// TIA Portal project "TFG_MaiteLopez" (V16)

(* hardware
DEVICE "S71500/ET200MP station_1"  S7-1500 station
   slot 0: "Perfil soporte_0"  Rack  6ES7 590-1***0-0AA0
   slot 1: "PLC_1"  CPU 1513-1 PN  6ES7 513-1AL01-0AB0  V2.8
      slot 3: "Display de la CPU_1"  6ES7591-1AA00-0AA0
      slot 32768: "Interfaz PROFINET_1"  X1
         slot 32769: "Puerto_1"  X1 P1
         slot 32770: "Puerto_2"  X1 P2
      slot 34817: "Virtual CP interface port_1"  Virtual CP interface port  Virtual CP interface port
DEVICE "HMI_1"  KTP400 Basic PN
   slot 0: "HMI_1"  KTP400 Basic PN  6AV2 123-2DB03-0AX0  16.0.0.0
   slot 1: "HMI_RT_1"  KTP400 Basic PN  6AV2 123-2DB03-0AX0  16.0.0.0
   slot 5: "HMI_1.IE_CP_1"  PROFINET Interface  16.0.0.0
      slot 1: "Interfaz PROFINET_1"  PROFINET Interface
         slot 1: "Port_1"  Port
*)

// ===== PLC "PLC_1"  CPU 1513-1 PN =====

VAR_GLOBAL   // PLC tag table "Entradas"
   "FactoryIO_Reseting" AT %I1.6 : Bool;
   "FactoryIO_Running" AT %I1.7 : Bool;
   "AtEntry" AT %I0.0 : Bool;
   "AtLoad" AT %I0.1 : Bool;
   "AtLeft" AT %I0.2 : Bool;
   "AtMiddle" AT %I0.3 : Bool;
   "AtRight" AT %I0.4 : Bool;
   "AtUnload" AT %I0.5 : Bool;
   "AtExit" AT %I0.6 : Bool;
   "MovingX" AT %I0.7 : Bool;
   "MovingZ" AT %I1.0 : Bool;
END_VAR

VAR_GLOBAL   // PLC tag table "HMI"
   "Marcha" AT %M5.0 : Bool;
   "Paro" AT %M5.1 : Bool;
   "Reset" AT %M5.2 : Bool;
   "AutoMan" AT %M5.3 : Bool;
   "Posicion" AT %MW8 : Int;
   "Men1" AT %M10.0 : Bool;
   "Men2" AT %M10.1 : Bool;
   "Men3" AT %M10.2 : Bool;
   "Emergencia" AT %M10.3 : Bool;
   "AuxMarcha" AT %M10.4 : Bool;
   "AuxParo" AT %M10.5 : Bool;
END_VAR

VAR_GLOBAL   // PLC tag table "Salidas"
   "TargetPosition" AT %QW2 : Word;
   "EntryConveyor" AT %Q0.0 : Bool;
   "LoadConveyor" AT %Q0.1 : Bool;
   "ForksLeft" AT %Q0.2 : Bool;
   "ForksRight" AT %Q0.3 : Bool;
   "Lift" AT %Q0.4 : Bool;
   "UnloadConveyor" AT %Q0.5 : Bool;
   "ExitConveyor" AT %Q0.6 : Bool;
   "Emitter" AT %Q1.2 : Bool;
   "Remover" AT %Q1.3 : Bool;
   "FactoryIO_Reset" AT %Q1.4 : Bool;
   "FactoryIO_Run" AT %Q1.5 : Bool;
END_VAR

VAR_GLOBAL   // PLC tag table "Señales de Control"
   "Inicio" AT %M0.0 : Bool;
   "SolCondIni" AT %M0.1 : Bool;
   "FinCondIni" AT %M0.2 : Bool;
   "ProdNorm" AT %M0.3 : Bool;
   "ParoFC" AT %M0.4 : Bool;
   "DejarCoger" AT %M0.5 : Bool;
   "FinDejar" AT %M0.7 : Bool;
   "InitGraf" AT %M1.6 : Bool;
   "ResetGraf" AT %M1.7 : Bool;
   "AuxInit" AT %M2.0 : Bool;
   "SolDejar" AT %M0.6 : Bool;
   "SolEntradaMaterial" AT %M1.2 : Bool;
   "FinEntradaMaterial" AT %M1.3 : Bool;
   "SolSalidaMaterial" AT %M1.4 : Bool;
   "FinSalidaMaterial" AT %M1.5 : Bool;
   "SolCoger" AT %M1.0 : Bool;
   "FinCoger" AT %M1.1 : Bool;
   "InicializarAlmacenOcupacion" AT %M2.1 : Bool;
END_VAR

DATA_BLOCK "Sensores"   // DB1
{ S7_Optimized_Access := 'FALSE' }
VERSION : 0.1
   VAR
      AlmacenOcupacion : Array[1..54] of Bool;
   END_VAR
BEGIN
END_DATA_BLOCK

DATA_BLOCK "CogerDejar_DB"   // DB2
{ S7_Optimized_Access := 'TRUE' }
VERSION : 0.1
// stored: InstanceOfName GCogerDejar
"GCogerDejar"
BEGIN
END_DATA_BLOCK

DATA_BLOCK "CondIniciales_DB"   // DB4
{ S7_Optimized_Access := 'TRUE' }
VERSION : 0.1
// stored: InstanceOfName GCondIniciales
"GCondIniciales"
BEGIN
END_DATA_BLOCK

DATA_BLOCK "MaterialIO_DB"   // DB5
{ S7_Optimized_Access := 'TRUE' }
VERSION : 0.1
// stored: InstanceOfName GMaterialIO
"GMaterialIO"
BEGIN
END_DATA_BLOCK

DATA_BLOCK "Emergencia_DB"   // DB6
{ S7_Optimized_Access := 'TRUE' }
VERSION : 0.1
// stored: InstanceOfName GEmergencia
"GEmergencia"
BEGIN
END_DATA_BLOCK

DATA_BLOCK "DB_OPCUA"   // DB7
{ S7_Optimized_Access := 'TRUE' }
VERSION : 0.1
   VAR
      control_parameters : Struct
         Control_Flag_New_Service : Bool := false;
         Control_Flag_Item_Completed : Bool;
         Control_Flag_Service_Completed : Bool;
      END_STRUCT;
      data_from_GW : Struct
         Id_Machine_Reference : UDInt;
         Id_Order_Reference : UDInt;
         Id_Batch_Reference : UDInt;
         Operation_Ref_Service_Type : UDInt := 1;
         Operation_No_of_Items : UDInt := 4;
      END_STRUCT;
      data_to_GW : Struct
         Id_Machine_Reference : UDInt;
         Id_Order_Reference : UDInt;
         Id_Batch_Reference : UDInt;
         Id_Ref_Service_Type : UDInt;
         Id_Item_Number : USInt;
         Data_Initial_Time_Stamp : String;
         Data_Final_Time_Stamp_1 : String;
         Data_Service_Time_Stamp : String;
      END_STRUCT;
   END_VAR
BEGIN
END_DATA_BLOCK

DATA_BLOCK "GestionarAlmacen_DB"   // DB8
{ S7_Optimized_Access := 'TRUE' }
VERSION : 0.1
// stored: InstanceOfName GGestionarAlmacen
"GGestionarAlmacen"
BEGIN
END_DATA_BLOCK

DATA_BLOCK "SecPrincipal_ST_DB"   // DB9
{ S7_Optimized_Access := 'TRUE' }
VERSION : 0.1
// stored: InstanceOfName GSecPrincipal_ST
"GSecPrincipal_ST"
BEGIN
END_DATA_BLOCK

// folder: System blocks/Program resources

DATA_BLOCK "IEC_Timer_0_DB"   // DB3
{ S7_Optimized_Access := 'TRUE' }
AUTHOR : Simatic
FAMILY : IEC
NAME : IEC_TMR
VERSION : 1.0
// stored: InstanceOfName IEC_TIMER
"IEC_TIMER"
BEGIN
END_DATA_BLOCK

DATA_BLOCK "Interfaz del cliente_1_Configuration"   // DB10
{ S7_Optimized_Access := 'TRUE' }
   VAR
      Connection : Struct
         ConnectInfo : OPC_UA_SessionConnectInfo;
         ConnectionHdl : DWord;
         ServerEndpointUrl : String[254] := 'opc.tcp://:4840';
      END_STRUCT;
      Namespaces : Struct
         NamespaceURIs : Array[0..0] of WString;
         ServerNamespaceIndexes : Array[0..0] of UInt;
         NamespaceStatusList : Array[0..0] of DWord;
         NamespaceCount : UInt := 0;
      END_STRUCT;
   END_VAR
BEGIN
   Connection.ConnectInfo.SessionName := WSTRING#'Conexión OPC UA_1';
   Connection.ConnectInfo.ApplicationName := WSTRING#'';
   Connection.ConnectInfo.SecurityMsgMode := 1;
   Connection.ConnectInfo.SecurityPolicy := 1;
   Connection.ConnectInfo.CheckServerCertificate := False;
   Connection.ConnectInfo.TransportProfile := 1;
   Connection.ConnectInfo.UserIdentityTokenType := 0;
   Connection.ConnectInfo.CertificateID := 0;
   Connection.ConnectInfo.SessionTimeout := T#30S;
   Connection.ConnectInfo.MonitorConnection := T#5S;
   Connection.ConnectInfo.LocaleIDs[0] := 'es-ES';
   Connection.ConnectInfo.LocaleIDs[1] := '';
   Connection.ConnectInfo.LocaleIDs[2] := '';
   Connection.ConnectInfo.LocaleIDs[3] := '';
   Connection.ConnectInfo.LocaleIDs[4] := '';
END_DATA_BLOCK

// folder: (top level)

FUNCTION_BLOCK "GGestionarAlmacen"   // FB1, GRAPH_PLUS
{ S7_Optimized_Access := 'TRUE' }
VERSION : 0.1
   VAR_INPUT
      OFF_SQ : Bool := false;   // Desactivar cadena
      INIT_SQ : Bool := false;   // Poner cadena en estado inicial
      ACK_EF : Bool := false;   // Acusar todos los errores y fallos
      S_PREV : Bool := false;   // Mostrar la etapa anterior en el parámetro S_NO
      S_NEXT : Bool := false;   // Mostrar la etapa siguiente en el parámetro S_NO
      SW_AUTO : Bool := false;   // Modo automático
      SW_TAP : Bool := false;   // Semiautomático/continuar con transición
      SW_TOP : Bool := false;   // Semiautomático/transición ignorada
      SW_MAN : Bool := false;   // Modo manual
      S_SEL : Int := 0;   // Seleccionar la etapa que debe mostrarse en S_NO
      S_ON : Bool := false;   // Activar la etapa del parámetro S_NO
      S_OFF : Bool := false;   // Desactivar el incremento presente en el parámetro S_NO
      T_PUSH : Bool := false;   // Habilitar conmutación de transición en modo semiautomático
   END_VAR
   VAR_OUTPUT
      S_NO : Int := 0;   // Número de etapa
      S_MORE : Bool := false;   // Existen más etapas que pueden mostrarse en S_NO.
      S_ACTIVE : Bool := false;   // El incremento presente en el parámetro S_NO está activo
      ERR_FLT : Bool := false;   // Error de grupo interlock o supervisión
      AUTO_ON : Bool := false;   // Modo automático activado
      TAP_ON : Bool := false;   // Modo semiautomático/etapa con transición activada
      TOP_ON : Bool := false;   // Modo semiautomático/Ignorar transición activado
      MAN_ON : Bool := false;   // Modo manual activado
   END_VAR
   VAR
      HMI_INFO : Array[0..8] of UInt;
      IF_PAR : G7_IfParPlus_V4;
      RT_DATA : G7_RTDataPlus_V4;   // Área de datos interna
      Trans1 : G7_TransitionPlus_V4;   // Estructura de la transición
      Trans2 : G7_TransitionPlus_V4;   // Estructura de la transición
      Trans3 : G7_TransitionPlus_V4;   // Estructura de la transición
      Trans4 : G7_TransitionPlus_V4;   // Estructura de la transición
      Trans5 : G7_TransitionPlus_V4;   // Estructura de la transición
      Trans6 : G7_TransitionPlus_V4;   // Estructura de la transición
      Trans7 : G7_TransitionPlus_V4;   // Estructura de la transición
      Trans8 : G7_TransitionPlus_V4;   // Estructura de la transición
      Trans9 : G7_TransitionPlus_V4;   // Estructura de la transición
      Trans10 : G7_TransitionPlus_V4;   // Estructura de la transición
      Trans11 : G7_TransitionPlus_V4;   // Estructura de la transición
      Trans12 : G7_TransitionPlus_V4;   // Estructura de la transición
      Trans14 : G7_TransitionPlus_V4;   // Estructura de la transición
      Trans18 : G7_TransitionPlus_V4;   // Estructura de la transición
      Trans19 : G7_TransitionPlus_V4;   // Estructura de la transición
      Trans26 : G7_TransitionPlus_V4;   // Estructura de la transición
      Trans27 : G7_TransitionPlus_V4;   // Estructura de la transición
      Trans28 : G7_TransitionPlus_V4;   // Estructura de la transición
      Trans29 : G7_TransitionPlus_V4;   // Estructura de la transición
      Trans30 : G7_TransitionPlus_V4;   // Estructura de la transición
      Trans31 : G7_TransitionPlus_V4;   // Estructura de la transición
      Trans32 : G7_TransitionPlus_V4;   // Estructura de la transición
      Trans35 : G7_TransitionPlus_V4;   // Estructura de la transición
      X40 : G7_StepPlus_V4;   // Estructura de la etapa
      X41 : G7_StepPlus_V4;   // Estructura de la etapa
      X42 : G7_StepPlus_V4;   // Estructura de la etapa
      X43 : G7_StepPlus_V4;   // Estructura de la etapa
      X44 : G7_StepPlus_V4;   // Estructura de la etapa
      X46 : G7_StepPlus_V4;   // Estructura de la etapa
      X47 : G7_StepPlus_V4;   // Estructura de la etapa
      X56 : G7_StepPlus_V4;   // Estructura de la etapa
      X57 : G7_StepPlus_V4;   // Estructura de la etapa
      X48 : G7_StepPlus_V4;   // Estructura de la etapa
      X49 : G7_StepPlus_V4;   // Estructura de la etapa
      X50 : G7_StepPlus_V4;   // Estructura de la etapa
      X52 : G7_StepPlus_V4;   // Estructura de la etapa
      X53 : G7_StepPlus_V4;   // Estructura de la etapa
      X54 : G7_StepPlus_V4;   // Estructura de la etapa
      X55 : G7_StepPlus_V4;   // Estructura de la etapa
      X51 : G7_StepPlus_V4;   // Estructura de la etapa
      X45 : G7_StepPlus_V4;   // Estructura de la etapa
      X58 : G7_StepPlus_V4;   // Estructura de la etapa
      SINI : Array[0..1] of USInt;
      LSTT : Array[0..22] of USInt;
      ATAJ : Array[0..22] of USInt;
      ATAB : Array[0..22] of USInt;
      PSTT : Array[0..22] of USInt;
      NSTT : Array[0..22] of USInt;
      ASSJ : Array[0..18] of USInt;
      ASSB : Array[0..18] of USInt;
      PTTS : Array[0..18] of USInt;
      NTTS : Array[0..18] of USInt;
      SW_SQTS : Array[0..18] of USInt;
      SWITCH : Array[0..6] of USInt;
      TVX : Array[0..8] of USInt;
      TTX : Array[0..8] of USInt;
      TSX : Array[0..1] of USInt;
      S00X : Array[0..1] of USInt;
      SOFFX : Array[0..1] of USInt;
      SONX : Array[0..1] of USInt;
      SAX : Array[0..1] of USInt;
      SERRX : Array[0..19] of USInt;
      SMX : Array[0..19] of USInt;
      S0X : Array[0..19] of USInt;
      S1X : Array[0..19] of USInt;
      IL_ALARM_INST : Diag_Alarm;
      SUP_ALARM_INST : Diag_Alarm;
      STEP_TIME_ALARM_INST : Diag_Alarm;
      IEC_TIMER_INST : IEC_TIMER;
      TRANSACTION_FLAG : Bool := false;
   END_VAR
   // SINI[0] := 2;
   // LSTT[0] := 255;
   // LSTT[1] := 255;
   // LSTT[2] := 255;
   // LSTT[3] := 255;
   // LSTT[4] := 255;
   // LSTT[5] := 255;
   // ATAJ[1] := 1;
   // ATAJ[2] := 2;
   // ATAJ[3] := 3;
   // ATAJ[4] := 4;
   // ATAJ[5] := 5;
   // ATAJ[6] := 6;
   // ATAB[1] := 7;
   // ATAB[2] := 8;
   // ATAB[3] := 12;
   // ATAB[4] := 4;
   // ATAB[5] := 5;
   // ATAB[6] := 6;
   // PSTT[1] := 1;
   // PSTT[2] := 2;
   // PSTT[3] := 3;
   // PSTT[4] := 4;
   // PSTT[5] := 5;
   // PSTT[6] := 6;
   // NSTT[0] := 1;
   // NSTT[1] := 2;
   // NSTT[2] := 3;
   // NSTT[3] := 4;
   // NSTT[4] := 17;
   // NSTT[5] := 6;
   // ASSJ[1] := 1;
   // ASSJ[2] := 2;
   // ASSJ[3] := 3;
   // ASSJ[4] := 4;
   // ASSJ[5] := 5;
   // ASSJ[6] := 6;
   // ASSB[1] := 1;
   // ASSB[2] := 2;
   // ASSB[3] := 3;
   // ASSB[4] := 4;
   // ASSB[5] := 5;
   // ASSB[6] := 6;
   // PTTS[0] := 255;
   // PTTS[2] := 1;
   // PTTS[3] := 2;
   // PTTS[4] := 3;
   // PTTS[5] := 21;
   // PTTS[6] := 5;
   // NTTS[1] := 1;
   // NTTS[2] := 2;
   // NTTS[3] := 3;
   // NTTS[4] := 4;
   // NTTS[5] := 5;
   // NTTS[6] := 6;
   // TVX[0] := 16#1;
   // TTX[0] := 16#1;
   // TSX[0] := 16#1;
   // S00X[0] := 16#1;
   // SOFFX[0] := 16#1;
   // SONX[0] := 16#1;
   // SAX[0] := 16#1;
   // SERRX[0] := 16#1;
   // SMX[0] := 16#1;
   // S0X[0] := 16#1;
   // S1X[0] := 16#1;
   // LSTT[6] := 255;
   // LSTT[8] := 255;
   // LSTT[9] := 255;
   // ATAJ[7] := 7;
   // ATAJ[8] := 8;
   // ATAJ[9] := 9;
   // ATAJ[10] := 10;
   // ATAJ[11] := 11;
   // ATAJ[12] := 12;
   // ATAB[7] := 1;
   // ATAB[8] := 9;
   // ATAB[9] := 2;
   // ATAB[10] := 10;
   // ATAB[11] := 11;
   // ATAB[12] := 3;
   // PSTT[7] := 1;
   // PSTT[8] := 2;
   // PSTT[9] := 2;
   // PSTT[10] := 7;
   // PSTT[11] := 8;
   // PSTT[12] := 3;
   // NSTT[6] := 9;
   // NSTT[8] := 7;
   // NSTT[9] := 8;
   // ASSJ[7] := 7;
   // ASSJ[8] := 8;
   // ASSJ[9] := 9;
   // ASSB[7] := 7;
   // ASSB[8] := 8;
   // ASSB[9] := 9;
   // PTTS[7] := 8;
   // PTTS[8] := 9;
   // PTTS[9] := 6;
   // NTTS[7] := 10;
   // NTTS[8] := 11;
   // NTTS[9] := 13;
   // SW_SQTS[2] := 1;
   // SW_SQTS[3] := 2;
   // SW_SQTS[4] := 3;
   // SW_SQTS[5] := 3;
   // SW_SQTS[6] := 3;
   // SW_SQTS[7] := 4;
   // SW_SQTS[8] := 5;
   // SW_SQTS[9] := 3;
   // LSTT[12] := 255;
   // LSTT[13] := 255;
   // LSTT[15] := 255;
   // ATAJ[13] := 13;
   // ATAJ[14] := 14;
   // ATAJ[15] := 15;
   // ATAJ[16] := 16;
   // ATAB[13] := 13;
   // ATAB[14] := 14;
   // ATAB[15] := 15;
   // ATAB[16] := 16;
   // PSTT[13] := 9;
   // PSTT[14] := 10;
   // PSTT[15] := 11;
   // PSTT[16] := 12;
   // SW_SQTS[15] := 6;
   // NSTT[12] := 11;
   // NSTT[13] := 10;
   // ASSB[13] := 13;
   // NSTT[15] := 16;
   // ASSB[12] := 12;
   // ASSJ[10] := 10;
   // ASSJ[11] := 11;
   // ASSJ[15] := 15;
   // ASSJ[14] := 14;
   // ASSB[10] := 10;
   // ASSB[11] := 11;
   // PSTT[19] := 15;
   // PSTT[18] := 14;
   // PTTS[10] := 13;
   // PTTS[11] := 12;
   // ATAJ[17] := 17;
   // NTTS[10] := 14;
   // NTTS[11] := 15;
   // SW_SQTS[10] := 3;
   // SW_SQTS[11] := 6;
   // SW_SQTS[14] := 6;
   // PTTS[15] := 18;
   // ASSJ[13] := 13;
   // PSTT[17] := 13;
   // LSTT[18] := 255;
   // SW_SQTS[13] := 6;
   // SW_SQTS[12] := 6;
   // NTTS[15] := 19;
   // NTTS[14] := 18;
   // NTTS[13] := 17;
   // NTTS[12] := 16;
   // PTTS[14] := 17;
   // PTTS[13] := 16;
   // PTTS[12] := 20;
   // ASSB[15] := 15;
   // ASSB[14] := 14;
   // ASSJ[12] := 12;
   // NSTT[18] := 15;
   // NSTT[17] := 14;
   // NSTT[16] := 13;
   // ATAB[19] := 19;
   // ATAB[18] := 18;
   // ATAB[17] := 17;
   // ATAJ[19] := 19;
   // ATAJ[18] := 18;
   // LSTT[17] := 255;
   // LSTT[16] := 255;
   // LSTT[20] := 255;
   // LSTT[21] := 255;
   // ATAJ[20] := 20;
   // ATAJ[21] := 21;
   // ATAB[20] := 20;
   // ATAB[21] := 21;
   // PSTT[20] := 16;
   // PSTT[21] := 17;
   // NSTT[20] := 12;
   // NSTT[21] := 5;
   // ASSJ[16] := 16;
   // ASSJ[17] := 17;
   // ASSB[16] := 16;
   // ASSB[17] := 17;
   // PTTS[16] := 15;
   // PTTS[17] := 4;
   // NTTS[16] := 20;
   // NTTS[17] := 21;
   // SW_SQTS[16] := 6;
   // SW_SQTS[17] := 3;
   // ATAJ[22] := 22;
   // ATAB[22] := 22;
   // PSTT[22] := 18;
   // LSTT[14] := 255;
   // NSTT[14] := 18;
   // ASSJ[18] := 18;
   // ASSB[18] := 18;
   // PTTS[18] := 14;
   // NTTS[18] := 22;
   // SW_SQTS[18] := 3;
BEGIN
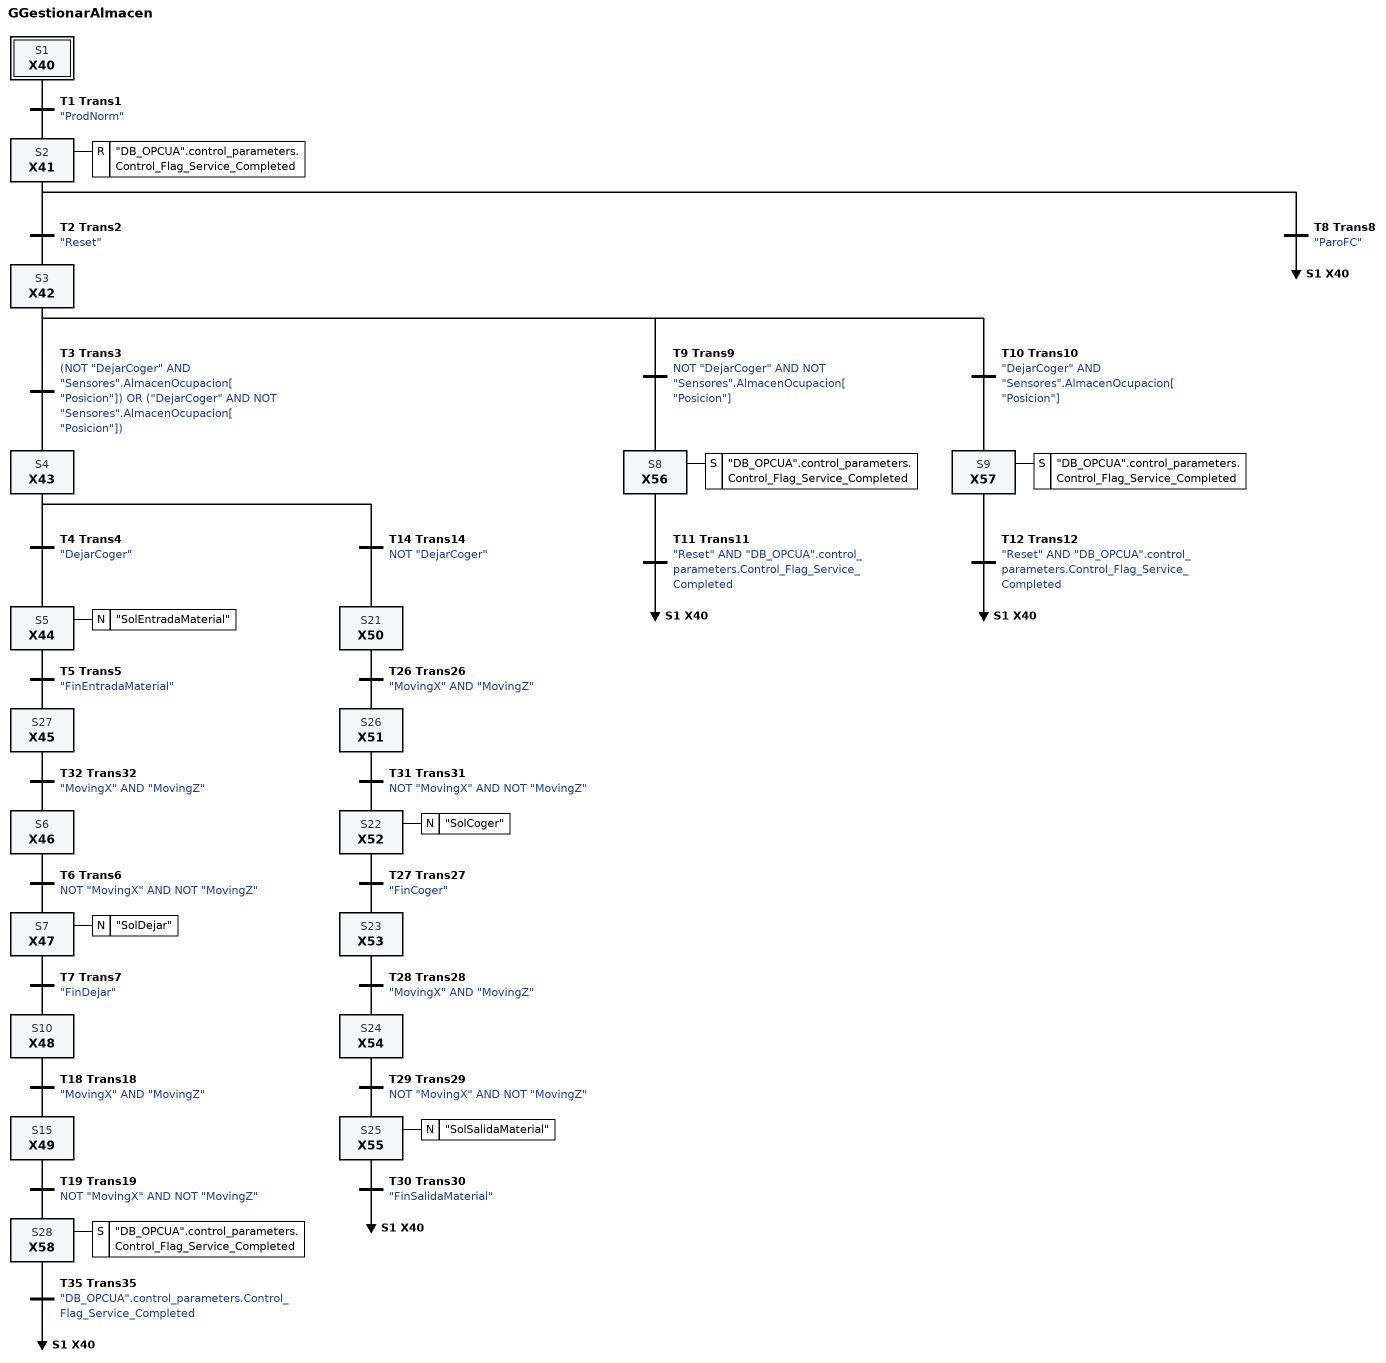
   // sequencer 1
   INITIAL_STEP X40:   // S1, max time T#10S, warning time T#7S
   END_STEP
   TRANSITION Trans1 FROM X40 TO X41   // T1
      := "ProdNorm";
   END_TRANSITION
   STEP X41:   // S2, max time T#10S, warning time T#7S
              R    "DB_OPCUA".control_parameters.Control_Flag_Service_Completed
   END_STEP
   TRANSITION Trans2 FROM X41 TO X42   // T2
      := "Reset";
   END_TRANSITION
   TRANSITION Trans8 FROM X41 TO X40   // T8, jump
      := "ParoFC";
   END_TRANSITION
   STEP X42:   // S3, max time T#10S, warning time T#7S
   END_STEP
   TRANSITION Trans3 FROM X42 TO X43   // T3
      := (NOT "DejarCoger" AND "Sensores".AlmacenOcupacion["Posicion"]) OR ("DejarCoger" AND NOT "Sensores".AlmacenOcupacion["Posicion"]);
   END_TRANSITION
   TRANSITION Trans9 FROM X42 TO X56   // T9
      := NOT "DejarCoger" AND NOT "Sensores".AlmacenOcupacion["Posicion"];
   END_TRANSITION
   TRANSITION Trans10 FROM X42 TO X57   // T10
      := "DejarCoger" AND "Sensores".AlmacenOcupacion["Posicion"];
   END_TRANSITION
   STEP X43:   // S4, max time T#10S, warning time T#7S
   END_STEP
   TRANSITION Trans4 FROM X43 TO X44   // T4
      := "DejarCoger";
   END_TRANSITION
   TRANSITION Trans14 FROM X43 TO X50   // T14
      := NOT "DejarCoger";
   END_TRANSITION
   STEP X44:   // S5, max time T#10S, warning time T#7S
              N    "SolEntradaMaterial"
   END_STEP
   TRANSITION Trans5 FROM X44 TO X45   // T5
      := "FinEntradaMaterial";
   END_TRANSITION
   STEP X46:   // S6, max time T#10S, warning time T#7S
   END_STEP
   TRANSITION Trans6 FROM X46 TO X47   // T6
      := NOT "MovingX" AND NOT "MovingZ";
   END_TRANSITION
   STEP X47:   // S7, max time T#10S, warning time T#7S
              N    "SolDejar"
   END_STEP
   TRANSITION Trans7 FROM X47 TO X48   // T7
      := "FinDejar";
   END_TRANSITION
   STEP X56:   // S8, max time T#10S, warning time T#7S
              S    "DB_OPCUA".control_parameters.Control_Flag_Service_Completed
   END_STEP
   TRANSITION Trans11 FROM X56 TO X40   // T11, jump
      := "Reset" AND "DB_OPCUA".control_parameters.Control_Flag_Service_Completed;
   END_TRANSITION
   STEP X57:   // S9, max time T#10S, warning time T#7S
              S    "DB_OPCUA".control_parameters.Control_Flag_Service_Completed
   END_STEP
   TRANSITION Trans12 FROM X57 TO X40   // T12, jump
      := "Reset" AND "DB_OPCUA".control_parameters.Control_Flag_Service_Completed;
   END_TRANSITION
   STEP X48:   // S10, max time T#10S, warning time T#7S
   END_STEP
   TRANSITION Trans18 FROM X48 TO X49   // T18
      := "MovingX" AND "MovingZ";
   END_TRANSITION
   STEP X49:   // S15, max time T#10S, warning time T#7S
   END_STEP
   TRANSITION Trans19 FROM X49 TO X58   // T19
      := NOT "MovingX" AND NOT "MovingZ";
   END_TRANSITION
   STEP X50:   // S21, max time T#10S, warning time T#7S
   END_STEP
   TRANSITION Trans26 FROM X50 TO X51   // T26
      := "MovingX" AND "MovingZ";
   END_TRANSITION
   STEP X55:   // S25, max time T#10S, warning time T#7S
              N    "SolSalidaMaterial"
   END_STEP
   TRANSITION Trans30 FROM X55 TO X40   // T30, jump
      := "FinSalidaMaterial";
   END_TRANSITION
   STEP X54:   // S24, max time T#10S, warning time T#7S
   END_STEP
   TRANSITION Trans29 FROM X54 TO X55   // T29
      := NOT "MovingX" AND NOT "MovingZ";
   END_TRANSITION
   STEP X53:   // S23, max time T#10S, warning time T#7S
   END_STEP
   TRANSITION Trans28 FROM X53 TO X54   // T28
      := "MovingX" AND "MovingZ";
   END_TRANSITION
   STEP X52:   // S22, max time T#10S, warning time T#7S
              N    "SolCoger"
   END_STEP
   TRANSITION Trans27 FROM X52 TO X53   // T27
      := "FinCoger";
   END_TRANSITION
   STEP X51:   // S26, max time T#10S, warning time T#7S
   END_STEP
   TRANSITION Trans31 FROM X51 TO X52   // T31
      := NOT "MovingX" AND NOT "MovingZ";
   END_TRANSITION
   STEP X45:   // S27, max time T#10S, warning time T#7S
   END_STEP
   TRANSITION Trans32 FROM X45 TO X46   // T32
      := "MovingX" AND "MovingZ";
   END_TRANSITION
   STEP X58:   // S28, max time T#10S, warning time T#7S
              S    "DB_OPCUA".control_parameters.Control_Flag_Service_Completed
   END_STEP
   TRANSITION Trans35 FROM X58 TO X40   // T35, jump
      := "DB_OPCUA".control_parameters.Control_Flag_Service_Completed;
   END_TRANSITION
END_FUNCTION_BLOCK

FUNCTION_BLOCK "GCondIniciales"   // FB2, GRAPH_PLUS
{ S7_Optimized_Access := 'TRUE' }
VERSION : 0.1
   VAR_INPUT
      SolCondIni : Bool;
      OFF_SQ : Bool := false;   // Desactivar cadena
      INIT_SQ : Bool := false;   // Poner cadena en estado inicial
      ACK_EF : Bool := false;   // Acusar todos los errores y fallos
      S_PREV : Bool := false;   // Mostrar la etapa anterior en el parámetro S_NO
      S_NEXT : Bool := false;   // Mostrar la etapa siguiente en el parámetro S_NO
      SW_AUTO : Bool := false;   // Modo automático
      SW_TAP : Bool := false;   // Semiautomático/continuar con transición
      SW_TOP : Bool := false;   // Semiautomático/transición ignorada
      SW_MAN : Bool := false;   // Modo manual
      S_SEL : Int := 0;   // Seleccionar la etapa que debe mostrarse en S_NO
      S_ON : Bool := false;   // Activar la etapa del parámetro S_NO
      S_OFF : Bool := false;   // Desactivar el incremento presente en el parámetro S_NO
      T_PUSH : Bool := false;   // Habilitar conmutación de transición en modo semiautomático
   END_VAR
   VAR_OUTPUT
      S_NO : Int := 0;   // Número de etapa
      S_MORE : Bool := false;   // Existen más etapas que pueden mostrarse en S_NO.
      S_ACTIVE : Bool := false;   // El incremento presente en el parámetro S_NO está activo
      ERR_FLT : Bool := false;   // Error de grupo interlock o supervisión
      AUTO_ON : Bool := false;   // Modo automático activado
      TAP_ON : Bool := false;   // Modo semiautomático/etapa con transición activada
      TOP_ON : Bool := false;   // Modo semiautomático/Ignorar transición activado
      MAN_ON : Bool := false;   // Modo manual activado
   END_VAR
   VAR
      HMI_INFO : Array[0..8] of UInt;
      IF_PAR : G7_IfParPlus_V4;
      RT_DATA : G7_RTDataPlus_V4;   // Área de datos interna
      Trans1 : G7_TransitionPlus_V4;   // Estructura de la transición
      Trans2 : G7_TransitionPlus_V4;   // Estructura de la transición
      Trans3 : G7_TransitionPlus_V4;   // Estructura de la transición
      Trans4 : G7_TransitionPlus_V4;   // Estructura de la transición
      Trans5 : G7_TransitionPlus_V4;   // Estructura de la transición
      X10 : G7_StepPlus_V4;   // Estructura de la etapa
      X11 : G7_StepPlus_V4;   // Estructura de la etapa
      X12 : G7_StepPlus_V4;   // Estructura de la etapa
      X14 : G7_StepPlus_V4;   // Estructura de la etapa
      X13 : G7_StepPlus_V4;   // Estructura de la etapa
      SINI : Array[0..1] of USInt;
      LSTT : Array[0..4] of USInt;
      ATAJ : Array[0..4] of USInt;
      ATAB : Array[0..4] of USInt;
      PSTT : Array[0..4] of USInt;
      NSTT : Array[0..4] of USInt;
      ASSJ : Array[0..4] of USInt;
      ASSB : Array[0..4] of USInt;
      PTTS : Array[0..4] of USInt;
      NTTS : Array[0..4] of USInt;
      SW_SQTS : Array[0..4] of USInt;
      SWITCH : Array[0..0] of USInt;
      TVX : Array[0..1] of USInt;
      TTX : Array[0..1] of USInt;
      TSX : Array[0..1] of USInt;
      S00X : Array[0..1] of USInt;
      SOFFX : Array[0..1] of USInt;
      SONX : Array[0..1] of USInt;
      SAX : Array[0..1] of USInt;
      SERRX : Array[0..5] of USInt;
      SMX : Array[0..5] of USInt;
      S0X : Array[0..5] of USInt;
      S1X : Array[0..5] of USInt;
      IL_ALARM_INST : Diag_Alarm;
      SUP_ALARM_INST : Diag_Alarm;
      STEP_TIME_ALARM_INST : Diag_Alarm;
      IEC_TIMER_INST : IEC_TIMER;
      TRANSACTION_FLAG : Bool := false;
   END_VAR
   // SINI[0] := 2;
   // LSTT[0] := 255;
   // LSTT[1] := 255;
   // ATAJ[1] := 1;
   // ATAJ[2] := 2;
   // ATAB[1] := 1;
   // ATAB[2] := 2;
   // PSTT[1] := 1;
   // PSTT[2] := 2;
   // NSTT[0] := 1;
   // NSTT[1] := 2;
   // ASSJ[1] := 1;
   // ASSJ[2] := 2;
   // ASSB[1] := 1;
   // ASSB[2] := 2;
   // PTTS[0] := 255;
   // PTTS[2] := 1;
   // NTTS[1] := 1;
   // NTTS[2] := 2;
   // TVX[0] := 16#1;
   // TTX[0] := 16#1;
   // TSX[0] := 16#1;
   // S00X[0] := 16#1;
   // SOFFX[0] := 16#1;
   // SONX[0] := 16#1;
   // SAX[0] := 16#1;
   // SERRX[0] := 16#1;
   // SMX[0] := 16#1;
   // S0X[0] := 16#1;
   // S1X[0] := 16#1;
   // LSTT[2] := 255;
   // ATAJ[3] := 3;
   // ATAB[3] := 3;
   // PSTT[3] := 3;
   // NSTT[2] := 4;
   // ASSJ[3] := 3;
   // ASSB[3] := 3;
   // PTTS[3] := 4;
   // NTTS[3] := 3;
   // LSTT[4] := 255;
   // ATAJ[4] := 4;
   // ATAB[4] := 4;
   // PSTT[4] := 4;
   // NSTT[4] := 3;
   // ASSJ[4] := 4;
   // ASSB[4] := 4;
   // PTTS[4] := 2;
   // NTTS[4] := 4;
BEGIN
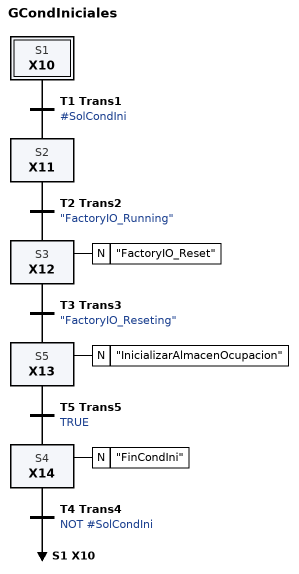
   // sequencer 1
   INITIAL_STEP X10:   // S1, max time T#10S, warning time T#7S
   END_STEP
   TRANSITION Trans1 FROM X10 TO X11   // T1
      := #SolCondIni;
   END_TRANSITION
   STEP X11:   // S2, max time T#10S, warning time T#7S
   END_STEP
   TRANSITION Trans2 FROM X11 TO X12   // T2
      := "FactoryIO_Running";
   END_TRANSITION
   STEP X12:   // S3, max time T#10S, warning time T#7S
              N    "FactoryIO_Reset"
   END_STEP
   TRANSITION Trans3 FROM X12 TO X13   // T3
      := "FactoryIO_Reseting";
   END_TRANSITION
   STEP X14:   // S4, max time T#10S, warning time T#7S
              N    "FinCondIni"
   END_STEP
   TRANSITION Trans4 FROM X14 TO X10   // T4, jump
      := NOT #SolCondIni;
   END_TRANSITION
   STEP X13:   // S5, max time T#10S, warning time T#7S
              N    "InicializarAlmacenOcupacion"
   END_STEP
   TRANSITION Trans5 FROM X13 TO X14   // T5
      := TRUE;
   END_TRANSITION
END_FUNCTION_BLOCK

FUNCTION_BLOCK "GMaterialIO"   // FB3, GRAPH_PLUS
{ S7_Optimized_Access := 'TRUE' }
VERSION : 0.1
   VAR_INPUT
      OFF_SQ : Bool := false;   // Desactivar cadena
      INIT_SQ : Bool := false;   // Poner cadena en estado inicial
      ACK_EF : Bool := false;   // Acusar todos los errores y fallos
      S_PREV : Bool := false;   // Mostrar la etapa anterior en el parámetro S_NO
      S_NEXT : Bool := false;   // Mostrar la etapa siguiente en el parámetro S_NO
      SW_AUTO : Bool := false;   // Modo automático
      SW_TAP : Bool := false;   // Semiautomático/continuar con transición
      SW_TOP : Bool := false;   // Semiautomático/transición ignorada
      SW_MAN : Bool := false;   // Modo manual
      S_SEL : Int := 0;   // Seleccionar la etapa que debe mostrarse en S_NO
      S_ON : Bool := false;   // Activar la etapa del parámetro S_NO
      S_OFF : Bool := false;   // Desactivar el incremento presente en el parámetro S_NO
      T_PUSH : Bool := false;   // Habilitar conmutación de transición en modo semiautomático
   END_VAR
   VAR_OUTPUT
      S_NO : Int := 0;   // Número de etapa
      S_MORE : Bool := false;   // Existen más etapas que pueden mostrarse en S_NO.
      S_ACTIVE : Bool := false;   // El incremento presente en el parámetro S_NO está activo
      ERR_FLT : Bool := false;   // Error de grupo interlock o supervisión
      AUTO_ON : Bool := false;   // Modo automático activado
      TAP_ON : Bool := false;   // Modo semiautomático/etapa con transición activada
      TOP_ON : Bool := false;   // Modo semiautomático/Ignorar transición activado
      MAN_ON : Bool := false;   // Modo manual activado
   END_VAR
   VAR
      HMI_INFO : Array[0..8] of UInt;
      IF_PAR : G7_IfParPlus_V6;
      RT_DATA : G7_RTDataPlus_V6;   // Área de datos interna
      Trans1 : G7_TransitionPlus_V6;   // Estructura de la transición
      Trans2 : G7_TransitionPlus_V6;   // Estructura de la transición
      Trans3 : G7_TransitionPlus_V6;   // Estructura de la transición
      Trans4 : G7_TransitionPlus_V6;   // Estructura de la transición
      Trans5 : G7_TransitionPlus_V6;   // Estructura de la transición
      Trans6 : G7_TransitionPlus_V6;   // Estructura de la transición
      Trans7 : G7_TransitionPlus_V6;   // Estructura de la transición
      Trans8 : G7_TransitionPlus_V6;   // Estructura de la transición
      Trans10 : G7_TransitionPlus_V6;   // Estructura de la transición
      Trans11 : G7_TransitionPlus_V6;   // Estructura de la transición
      Trans12 : G7_TransitionPlus_V6;   // Estructura de la transición
      Trans13 : G7_TransitionPlus_V6;   // Estructura de la transición
      Trans14 : G7_TransitionPlus_V6;   // Estructura de la transición
      Trans15 : G7_TransitionPlus_V6;   // Estructura de la transición
      Trans16 : G7_TransitionPlus_V6;   // Estructura de la transición
      X80 : G7_StepPlus_V6;   // Estructura de la etapa
      X81 : G7_StepPlus_V6;   // Estructura de la etapa
      X82 : G7_StepPlus_V6;   // Estructura de la etapa
      X83 : G7_StepPlus_V6;   // Estructura de la etapa
      X84 : G7_StepPlus_V6;   // Estructura de la etapa
      X85 : G7_StepPlus_V6;   // Estructura de la etapa
      X86 : G7_StepPlus_V6;   // Estructura de la etapa
      X87 : G7_StepPlus_V6;   // Estructura de la etapa
      X88 : G7_StepPlus_V6;   // Estructura de la etapa
      X89 : G7_StepPlus_V6;   // Estructura de la etapa
      X91 : G7_StepPlus_V6;   // Estructura de la etapa
      X92 : G7_StepPlus_V6;   // Estructura de la etapa
      X90 : G7_StepPlus_V6;   // Estructura de la etapa
      X93 : G7_StepPlus_V6;   // Estructura de la etapa
      SINI : Array[0..1] of USInt;
      LSTT : Array[0..14] of USInt;
      ATAJ : Array[0..14] of USInt;
      ATAB : Array[0..14] of USInt;
      PSTT : Array[0..14] of USInt;
      NSTT : Array[0..14] of USInt;
      ASSJ : Array[0..13] of USInt;
      ASSB : Array[0..13] of USInt;
      PTTS : Array[0..13] of USInt;
      NTTS : Array[0..13] of USInt;
      SW_SQTS : Array[0..13] of USInt;
      SWITCH : Array[0..1] of USInt;
      TVX : Array[0..3] of USInt;
      TTX : Array[0..3] of USInt;
      TSX : Array[0..1] of USInt;
      S00X : Array[0..1] of USInt;
      SOFFX : Array[0..1] of USInt;
      SONX : Array[0..1] of USInt;
      SAX : Array[0..1] of USInt;
      SERRX : Array[0..14] of USInt;
      SMX : Array[0..14] of USInt;
      S0X : Array[0..14] of USInt;
      S1X : Array[0..14] of USInt;
      IL_ALARM_INST : Diag_Alarm;
      SUP_ALARM_INST : Diag_Alarm;
      STEP_TIME_ALARM_INST : Diag_Alarm;
      IEC_TIMER_INST : IEC_TIMER;
      TRANSACTION_FLAG : Bool := false;
   END_VAR
   // SINI[0] := 2;
   // LSTT[0] := 255;
   // LSTT[1] := 255;
   // LSTT[2] := 255;
   // LSTT[3] := 255;
   // LSTT[4] := 255;
   // LSTT[5] := 255;
   // ATAJ[1] := 1;
   // ATAJ[2] := 2;
   // ATAJ[3] := 3;
   // ATAJ[4] := 4;
   // ATAJ[5] := 5;
   // ATAJ[6] := 6;
   // ATAB[1] := 1;
   // ATAB[2] := 2;
   // ATAB[3] := 3;
   // ATAB[4] := 4;
   // ATAB[5] := 5;
   // ATAB[6] := 6;
   // PSTT[1] := 1;
   // PSTT[2] := 2;
   // PSTT[3] := 3;
   // PSTT[4] := 4;
   // PSTT[5] := 5;
   // PSTT[6] := 6;
   // NSTT[0] := 1;
   // NSTT[1] := 2;
   // NSTT[2] := 3;
   // NSTT[3] := 4;
   // NSTT[4] := 5;
   // NSTT[5] := 6;
   // ASSJ[1] := 1;
   // ASSJ[2] := 2;
   // ASSJ[3] := 3;
   // ASSJ[4] := 4;
   // ASSJ[5] := 5;
   // ASSJ[6] := 6;
   // ASSB[1] := 1;
   // ASSB[2] := 2;
   // ASSB[3] := 3;
   // ASSB[4] := 4;
   // ASSB[5] := 5;
   // ASSB[6] := 6;
   // PTTS[0] := 255;
   // PTTS[2] := 1;
   // PTTS[3] := 2;
   // PTTS[4] := 3;
   // PTTS[5] := 4;
   // PTTS[6] := 5;
   // NTTS[1] := 1;
   // NTTS[2] := 2;
   // NTTS[3] := 3;
   // NTTS[4] := 4;
   // NTTS[5] := 5;
   // NTTS[6] := 6;
   // TVX[0] := 16#1;
   // TTX[0] := 16#1;
   // TSX[0] := 16#1;
   // S00X[0] := 16#1;
   // SOFFX[0] := 16#1;
   // SONX[0] := 16#1;
   // SAX[0] := 16#1;
   // SERRX[0] := 16#1;
   // SMX[0] := 16#1;
   // S0X[0] := 16#1;
   // S1X[0] := 16#1;
   // LSTT[7] := 255;
   // LSTT[8] := 255;
   // LSTT[9] := 255;
   // LSTT[10] := 255;
   // LSTT[11] := 255;
   // LSTT[13] := 255;
   // ATAJ[7] := 7;
   // ATAJ[8] := 8;
   // ATAJ[9] := 9;
   // ATAJ[10] := 10;
   // ATAJ[11] := 11;
   // ATAJ[12] := 12;
   // ATAJ[13] := 13;
   // ATAB[0] := 7;
   // ATAB[8] := 8;
   // ATAB[9] := 9;
   // ATAB[10] := 10;
   // ATAB[11] := 11;
   // ATAB[12] := 12;
   // ATAB[13] := 13;
   // PSTT[8] := 7;
   // PSTT[9] := 8;
   // PSTT[10] := 9;
   // PSTT[11] := 10;
   // PSTT[12] := 11;
   // PSTT[13] := 12;
   // NSTT[7] := 7;
   // NSTT[8] := 8;
   // NSTT[9] := 9;
   // NSTT[10] := 12;
   // NSTT[11] := 11;
   // NSTT[13] := 10;
   // ASSJ[7] := 7;
   // ASSJ[8] := 8;
   // ASSJ[9] := 9;
   // ASSJ[10] := 10;
   // ASSJ[11] := 11;
   // ASSJ[12] := 12;
   // ASSB[7] := 7;
   // ASSB[8] := 8;
   // ASSB[9] := 9;
   // ASSB[10] := 10;
   // ASSB[11] := 11;
   // ASSB[12] := 12;
   // PTTS[7] := 7;
   // PTTS[8] := 8;
   // PTTS[9] := 9;
   // PTTS[10] := 13;
   // PTTS[11] := 11;
   // PTTS[12] := 10;
   // NTTS[7] := 8;
   // NTTS[8] := 9;
   // NTTS[9] := 10;
   // NTTS[10] := 11;
   // NTTS[11] := 12;
   // NTTS[12] := 13;
   // SW_SQTS[1] := 1;
   // SW_SQTS[2] := 1;
   // SW_SQTS[3] := 1;
   // SW_SQTS[4] := 1;
   // SW_SQTS[5] := 1;
   // SW_SQTS[6] := 1;
   // SW_SQTS[7] := 2;
   // SW_SQTS[8] := 2;
   // SW_SQTS[9] := 2;
   // SW_SQTS[10] := 2;
   // SW_SQTS[11] := 2;
   // SW_SQTS[12] := 2;
   // LSTT[12] := 255;
   // ATAJ[14] := 14;
   // ATAB[14] := 14;
   // PSTT[14] := 13;
   // NSTT[12] := 13;
   // ASSJ[13] := 13;
   // ASSB[13] := 13;
   // PTTS[13] := 12;
   // NTTS[13] := 14;
   // SW_SQTS[13] := 2;
BEGIN
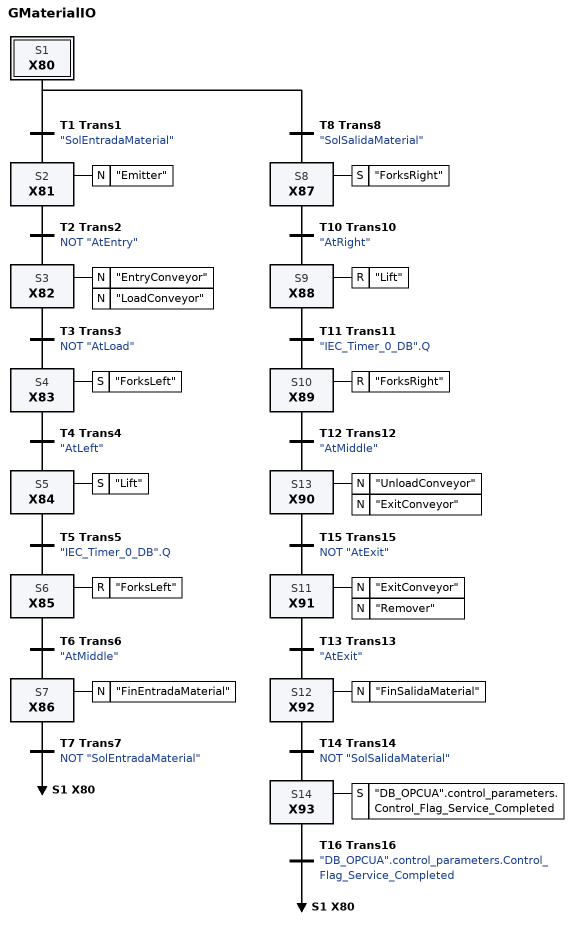
   // sequencer 1
   INITIAL_STEP X80:   // S1, max time T#10S, warning time T#7S
   END_STEP
   TRANSITION Trans1 FROM X80 TO X81   // T1
      := "SolEntradaMaterial";
   END_TRANSITION
   TRANSITION Trans8 FROM X80 TO X87   // T8
      := "SolSalidaMaterial";
   END_TRANSITION
   STEP X81:   // S2, max time T#10S, warning time T#7S
              N    "Emitter"
   END_STEP
   TRANSITION Trans2 FROM X81 TO X82   // T2
      := NOT "AtEntry";
   END_TRANSITION
   STEP X82:   // S3, max time T#10S, warning time T#7S
              N    "EntryConveyor"
              N    "LoadConveyor"
   END_STEP
   TRANSITION Trans3 FROM X82 TO X83   // T3
      := NOT "AtLoad";
   END_TRANSITION
   STEP X83:   // S4, max time T#10S, warning time T#7S
              S    "ForksLeft"
   END_STEP
   TRANSITION Trans4 FROM X83 TO X84   // T4
      := "AtLeft";
   END_TRANSITION
   STEP X84:   // S5, max time T#10S, warning time T#7S
              S    "Lift"
   END_STEP
   TRANSITION Trans5 FROM X84 TO X85   // T5
      := "IEC_Timer_0_DB".Q;
   END_TRANSITION
   STEP X85:   // S6, max time T#10S, warning time T#7S
              R    "ForksLeft"
   END_STEP
   TRANSITION Trans6 FROM X85 TO X86   // T6
      := "AtMiddle";
   END_TRANSITION
   STEP X86:   // S7, max time T#10S, warning time T#7S
              N    "FinEntradaMaterial"
   END_STEP
   TRANSITION Trans7 FROM X86 TO X80   // T7, jump
      := NOT "SolEntradaMaterial";
   END_TRANSITION
   STEP X87:   // S8, max time T#10S, warning time T#7S
              S    "ForksRight"
   END_STEP
   TRANSITION Trans10 FROM X87 TO X88   // T10
      := "AtRight";
   END_TRANSITION
   STEP X88:   // S9, max time T#10S, warning time T#7S
              R    "Lift"
   END_STEP
   TRANSITION Trans11 FROM X88 TO X89   // T11
      := "IEC_Timer_0_DB".Q;
   END_TRANSITION
   STEP X89:   // S10, max time T#10S, warning time T#7S
              R    "ForksRight"
   END_STEP
   TRANSITION Trans12 FROM X89 TO X90   // T12
      := "AtMiddle";
   END_TRANSITION
   STEP X91:   // S11, max time T#10S, warning time T#7S
              N    "ExitConveyor"
              N    "Remover"
   END_STEP
   TRANSITION Trans13 FROM X91 TO X92   // T13
      := "AtExit";
   END_TRANSITION
   STEP X92:   // S12, max time T#10S, warning time T#7S
              N    "FinSalidaMaterial"
   END_STEP
   TRANSITION Trans14 FROM X92 TO X93   // T14
      := NOT "SolSalidaMaterial";
   END_TRANSITION
   STEP X90:   // S13, max time T#10S, warning time T#7S
              N    "UnloadConveyor"
              N    "ExitConveyor"
   END_STEP
   TRANSITION Trans15 FROM X90 TO X91   // T15
      := NOT "AtExit";
   END_TRANSITION
   STEP X93:   // S14, max time T#10S, warning time T#7S
              S    "DB_OPCUA".control_parameters.Control_Flag_Service_Completed
   END_STEP
   TRANSITION Trans16 FROM X93 TO X80   // T16, jump
      := "DB_OPCUA".control_parameters.Control_Flag_Service_Completed;
   END_TRANSITION
END_FUNCTION_BLOCK

FUNCTION_BLOCK "GCogerDejar"   // FB4, GRAPH_PLUS
{ S7_Optimized_Access := 'TRUE' }
VERSION : 0.1
   VAR_INPUT
      OFF_SQ : Bool := false;   // Desactivar cadena
      INIT_SQ : Bool := false;   // Poner cadena en estado inicial
      ACK_EF : Bool := false;   // Acusar todos los errores y fallos
      S_PREV : Bool := false;   // Mostrar la etapa anterior en el parámetro S_NO
      S_NEXT : Bool := false;   // Mostrar la etapa siguiente en el parámetro S_NO
      SW_AUTO : Bool := false;   // Modo automático
      SW_TAP : Bool := false;   // Semiautomático/continuar con transición
      SW_TOP : Bool := false;   // Semiautomático/transición ignorada
      SW_MAN : Bool := false;   // Modo manual
      S_SEL : Int := 0;   // Seleccionar la etapa que debe mostrarse en S_NO
      S_ON : Bool := false;   // Activar la etapa del parámetro S_NO
      S_OFF : Bool := false;   // Desactivar el incremento presente en el parámetro S_NO
      T_PUSH : Bool := false;   // Habilitar conmutación de transición en modo semiautomático
   END_VAR
   VAR_OUTPUT
      S_NO : Int := 0;   // Número de etapa
      S_MORE : Bool := false;   // Existen más etapas que pueden mostrarse en S_NO.
      S_ACTIVE : Bool := false;   // El incremento presente en el parámetro S_NO está activo
      ERR_FLT : Bool := false;   // Error de grupo interlock o supervisión
      AUTO_ON : Bool := false;   // Modo automático activado
      TAP_ON : Bool := false;   // Modo semiautomático/etapa con transición activada
      TOP_ON : Bool := false;   // Modo semiautomático/Ignorar transición activado
      MAN_ON : Bool := false;   // Modo manual activado
   END_VAR
   VAR
      HMI_INFO : Array[0..8] of UInt;
      IF_PAR : G7_IfParPlus_V4;
      RT_DATA : G7_RTDataPlus_V4;   // Área de datos interna
      Trans1 : G7_TransitionPlus_V4;   // Estructura de la transición
      Trans7 : G7_TransitionPlus_V4;   // Estructura de la transición
      Trans9 : G7_TransitionPlus_V4;   // Estructura de la transición
      Trans10 : G7_TransitionPlus_V4;   // Estructura de la transición
      Trans11 : G7_TransitionPlus_V4;   // Estructura de la transición
      Trans12 : G7_TransitionPlus_V4;   // Estructura de la transición
      Trans14 : G7_TransitionPlus_V4;   // Estructura de la transición
      Trans15 : G7_TransitionPlus_V4;   // Estructura de la transición
      Trans16 : G7_TransitionPlus_V4;   // Estructura de la transición
      Trans17 : G7_TransitionPlus_V4;   // Estructura de la transición
      Trans18 : G7_TransitionPlus_V4;   // Estructura de la transición
      Trans19 : G7_TransitionPlus_V4;   // Estructura de la transición
      X60 : G7_StepPlus_V4;   // Estructura de la etapa
      X69 : G7_StepPlus_V4;   // Estructura de la etapa
      X66 : G7_StepPlus_V4;   // Estructura de la etapa
      X67 : G7_StepPlus_V4;   // Estructura de la etapa
      X61 : G7_StepPlus_V4;   // Estructura de la etapa
      X62 : G7_StepPlus_V4;   // Estructura de la etapa
      X70 : G7_StepPlus_V4;   // Estructura de la etapa
      X63 : G7_StepPlus_V4;   // Estructura de la etapa
      X64 : G7_StepPlus_V4;   // Estructura de la etapa
      X68 : G7_StepPlus_V4;   // Estructura de la etapa
      X65 : G7_StepPlus_V4;   // Estructura de la etapa
      SINI : Array[0..1] of USInt;
      LSTT : Array[0..11] of USInt;
      ATAJ : Array[0..11] of USInt;
      ATAB : Array[0..11] of USInt;
      PSTT : Array[0..11] of USInt;
      NSTT : Array[0..11] of USInt;
      ASSJ : Array[0..10] of USInt;
      ASSB : Array[0..10] of USInt;
      PTTS : Array[0..10] of USInt;
      NTTS : Array[0..10] of USInt;
      SW_SQTS : Array[0..10] of USInt;
      SWITCH : Array[0..1] of USInt;
      TVX : Array[0..3] of USInt;
      TTX : Array[0..3] of USInt;
      TSX : Array[0..1] of USInt;
      S00X : Array[0..1] of USInt;
      SOFFX : Array[0..1] of USInt;
      SONX : Array[0..1] of USInt;
      SAX : Array[0..1] of USInt;
      SERRX : Array[0..11] of USInt;
      SMX : Array[0..11] of USInt;
      S0X : Array[0..11] of USInt;
      S1X : Array[0..11] of USInt;
      IL_ALARM_INST : Diag_Alarm;
      SUP_ALARM_INST : Diag_Alarm;
      STEP_TIME_ALARM_INST : Diag_Alarm;
      IEC_TIMER_INST : IEC_TIMER;
      TRANSACTION_FLAG : Bool := false;
   END_VAR
   // ATAJ[8] := 8;
   // LSTT[8] := 255;
   // SINI[0] := 2;
   // LSTT[0] := 255;
   // LSTT[1] := 255;
   // LSTT[2] := 255;
   // LSTT[6] := 255;
   // ATAJ[1] := 1;
   // ATAJ[2] := 2;
   // ATAJ[3] := 3;
   // ATAJ[4] := 4;
   // ATAB[1] := 1;
   // ATAB[2] := 2;
   // ATAB[3] := 3;
   // ATAB[4] := 4;
   // PSTT[2] := 5;
   // PSTT[3] := 10;
   // PSTT[4] := 7;
   // NSTT[0] := 4;
   // NSTT[1] := 5;
   // NSTT[2] := 7;
   // NSTT[6] := 6;
   // ASSJ[1] := 1;
   // ASSJ[2] := 2;
   // ASSJ[3] := 3;
   // ASSB[1] := 1;
   // ASSB[2] := 2;
   // ASSB[3] := 3;
   // PTTS[0] := 255;
   // PTTS[2] := 11;
   // PTTS[3] := 7;
   // NTTS[1] := 6;
   // NTTS[2] := 7;
   // NTTS[3] := 8;
   // SW_SQTS[7] := 2;
   // SW_SQTS[2] := 1;
   // SW_SQTS[3] := 1;
   // TVX[0] := 16#1;
   // TTX[0] := 16#1;
   // TSX[0] := 16#1;
   // S00X[0] := 16#1;
   // SOFFX[0] := 16#1;
   // SONX[0] := 16#1;
   // SAX[0] := 16#1;
   // SERRX[0] := 16#1;
   // SMX[0] := 16#1;
   // S0X[0] := 16#1;
   // S1X[0] := 16#1;
   // LSTT[4] := 255;
   // LSTT[5] := 255;
   // ATAJ[5] := 5;
   // ATAJ[6] := 6;
   // ATAB[5] := 5;
   // ATAB[6] := 6;
   // PSTT[5] := 8;
   // PSTT[6] := 1;
   // NSTT[4] := 8;
   // NSTT[5] := 10;
   // ASSJ[4] := 4;
   // ASSJ[5] := 5;
   // ASSB[4] := 4;
   // ASSB[5] := 5;
   // PTTS[5] := 1;
   // NTTS[4] := 1;
   // NTTS[5] := 2;
   // SW_SQTS[4] := 2;
   // SW_SQTS[5] := 2;
   // LSTT[7] := 255;
   // ATAJ[7] := 7;
   // ATAB[7] := 7;
   // PSTT[7] := 2;
   // NSTT[7] := 3;
   // ASSJ[6] := 6;
   // ASSB[6] := 6;
   // PTTS[6] := 6;
   // NTTS[6] := 10;
   // SW_SQTS[6] := 1;
   // ATAB[8] := 8;
   // PSTT[1] := 4;
   // PSTT[8] := 3;
   // NSTT[8] := 9;
   // ASSJ[7] := 7;
   // ASSB[7] := 7;
   // PTTS[7] := 2;
   // NTTS[7] := 4;
   // LSTT[9] := 255;
   // LSTT[11] := 255;
   // ATAJ[9] := 9;
   // ATAJ[10] := 10;
   // ATAJ[11] := 11;
   // ATAB[9] := 9;
   // ATAB[10] := 10;
   // PSTT[9] := 9;
   // PSTT[10] := 6;
   // NSTT[9] := 1;
   // NSTT[11] := 2;
   // ASSJ[8] := 8;
   // ASSJ[9] := 9;
   // ASSJ[10] := 10;
   // ASSB[8] := 8;
   // ASSB[9] := 9;
   // ASSB[10] := 10;
   // PTTS[8] := 4;
   // PTTS[9] := 8;
   // PTTS[10] := 5;
   // NTTS[8] := 5;
   // NTTS[9] := 9;
   // NTTS[10] := 3;
   // SW_SQTS[8] := 2;
   // SW_SQTS[9] := 1;
   // SW_SQTS[10] := 2;
   // ATAB[0] := 11;
   // PTTS[1] := 9;
   // SW_SQTS[1] := 1;
BEGIN
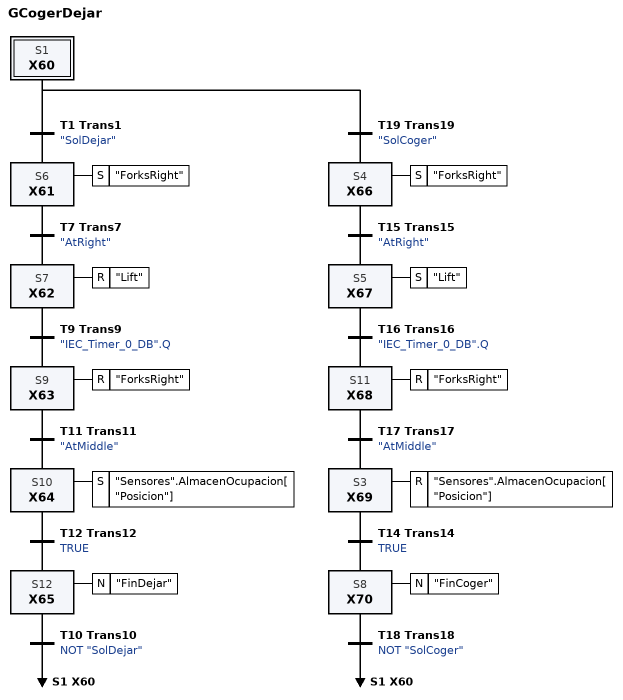
   // sequencer 1
   INITIAL_STEP X60:   // S1, max time T#10S, warning time T#7S
   END_STEP
   TRANSITION Trans1 FROM X60 TO X61   // T1
      := "SolDejar";
   END_TRANSITION
   TRANSITION Trans19 FROM X60 TO X66   // T19
      := "SolCoger";
   END_TRANSITION
   STEP X61:   // S6, max time T#10S, warning time T#7S
              S    "ForksRight"
   END_STEP
   TRANSITION Trans7 FROM X61 TO X62   // T7
      := "AtRight";
   END_TRANSITION
   STEP X62:   // S7, max time T#10S, warning time T#7S
              R    "Lift"
   END_STEP
   TRANSITION Trans9 FROM X62 TO X63   // T9
      := "IEC_Timer_0_DB".Q;
   END_TRANSITION
   STEP X65:   // S12, max time T#10S, warning time T#7S
              N    "FinDejar"
   END_STEP
   TRANSITION Trans10 FROM X65 TO X60   // T10, jump
      := NOT "SolDejar";
   END_TRANSITION
   STEP X63:   // S9, max time T#10S, warning time T#7S
              R    "ForksRight"
   END_STEP
   TRANSITION Trans11 FROM X63 TO X64   // T11
      := "AtMiddle";
   END_TRANSITION
   STEP X64:   // S10, max time T#10S, warning time T#7S
              S    "Sensores".AlmacenOcupacion["Posicion"]
   END_STEP
   TRANSITION Trans12 FROM X64 TO X65   // T12
      := TRUE;
   END_TRANSITION
   STEP X69:   // S3, max time T#10S, warning time T#7S
              R    "Sensores".AlmacenOcupacion["Posicion"]
   END_STEP
   TRANSITION Trans14 FROM X69 TO X70   // T14
      := TRUE;
   END_TRANSITION
   STEP X66:   // S4, max time T#10S, warning time T#7S
              S    "ForksRight"
   END_STEP
   TRANSITION Trans15 FROM X66 TO X67   // T15
      := "AtRight";
   END_TRANSITION
   STEP X67:   // S5, max time T#10S, warning time T#7S
              S    "Lift"
   END_STEP
   TRANSITION Trans16 FROM X67 TO X68   // T16
      := "IEC_Timer_0_DB".Q;
   END_TRANSITION
   STEP X68:   // S11, max time T#10S, warning time T#7S
              R    "ForksRight"
   END_STEP
   TRANSITION Trans17 FROM X68 TO X69   // T17
      := "AtMiddle";
   END_TRANSITION
   STEP X70:   // S8, max time T#10S, warning time T#7S
              N    "FinCoger"
   END_STEP
   TRANSITION Trans18 FROM X70 TO X60   // T18, jump
      := NOT "SolCoger";
   END_TRANSITION
END_FUNCTION_BLOCK

FUNCTION_BLOCK "GSecPrincipal_ST"   // FB5, SCL
{ S7_Optimized_Access := 'TRUE' }
VERSION : 0.1
   VAR_INPUT
      Init : Bool;
      Reset : Bool;
      SolModoAuto : Bool;
      SolParoFC : Bool;
      FinCondIni : Bool := true;
      FinMarchaPre : Bool := true;
      FinProces : Bool;
      FinMarchaFin : Bool := true;
   END_VAR
   VAR_OUTPUT
      Inicio : Bool;
      SolCondIni : Bool := false;
      SolMarchaPre : Bool := false;
      ProdNorm : Bool;
      ParoFC : Bool;
      SolMarchaFin : Bool := false;
   END_VAR
   VAR
      X0 : Bool;
      X1 : Bool;
      X2 : Bool;
      X3 : Bool;
      X4 : Bool;
      X5 : Bool;
   END_VAR
BEGIN
   (*________________________________________________________________________

   SecPrincipal: Organiza tanto el arranque del sistema en modo automático 
   como la parada programada del mismo.
   ________________________________________________________________________ *)

   (* PARTE SECUENCIAL *)
   (* Set -Reset _______________________________________________________ X0 *)
   IF ((#X5 AND #FinMarchaFin) OR #Init) THEN
       #X0 := 1;
   END_IF;
   IF (#X1 OR #Reset) THEN
       #X0 := 0;
   END_IF;

   (* Set -Reset ________________________________________________________________ X1 *)
   IF ((#X0 AND "Marcha")) THEN
       #X1 := 1;
   END_IF;
   IF (#X2 OR #Init OR #Reset) THEN
       #X1 := 0;
   END_IF;

   (* Set -Reset ________________________________________________________________ X2 *)
   IF ((#X1 AND #FinCondIni)) THEN
       #X2 := 1;
   END_IF;
   IF (#X3 OR #Init OR #Reset) THEN
       #X2 := 0;
   END_IF;

   (* Set -Reset ________________________________________________________________ X3 *)
   IF (#X2 AND #FinMarchaPre) THEN
       #X3 := 1;
   END_IF;
   IF (#X4 OR #Init OR #Reset) THEN
       #X3 := 0;
   END_IF;

   (* Set -Reset ________________________________________________________________ X4 *)
   IF ((#X3 AND #SolParoFC)) THEN
       #X4 := 1;
   END_IF;
   IF (#X5 OR #Init OR #Reset) THEN
       #X4 := 0;
   END_IF;

   (* Set -Reset ________________________________________________________________ X5 *)
   IF ((#X4 AND #FinProces)) THEN
       #X5 := 1;
   END_IF;
   IF (#X0 OR #Init OR #Reset) THEN
       #X5 := 0;
   END_IF;

   (*________________________________________________________________________
   SecPrincipal: señales de mando que informan a producción normal sobre 
   el estado del sistema en cada momento
   ________________________________________________________________________ *)
   (* PARTE COMBINACIONAL *)
   #Inicio         := #X0;
   #SolCondIni     := #X1;
   #SolMarchaPre   := #X2;
   #ProdNorm       := #X3;
   #ParoFC         := #X4;
   #SolMarchaFin   := #X5;
END_FUNCTION_BLOCK

FUNCTION_BLOCK "GEmergencia"   // FB6, GRAPH_PLUS
{ S7_Optimized_Access := 'TRUE' }
VERSION : 0.1
   VAR_INPUT
      SolEmergencia : Bool;
      SolParoEmergencia : Bool;
      Inicio : Bool;
      OFF_SQ : Bool := false;   // Desactivar cadena
      INIT_SQ : Bool := false;   // Poner cadena en estado inicial
      ACK_EF : Bool := false;   // Acusar todos los errores y fallos
      S_PREV : Bool := false;   // Mostrar la etapa anterior en el parámetro S_NO
      S_NEXT : Bool := false;   // Mostrar la etapa siguiente en el parámetro S_NO
      SW_AUTO : Bool := false;   // Modo automático
      SW_TAP : Bool := false;   // Semiautomático/continuar con transición
      SW_TOP : Bool := false;   // Semiautomático/transición ignorada
      SW_MAN : Bool := false;   // Modo manual
      S_SEL : Int := 0;   // Seleccionar la etapa que debe mostrarse en S_NO
      S_ON : Bool := false;   // Activar la etapa del parámetro S_NO
      S_OFF : Bool := false;   // Desactivar el incremento presente en el parámetro S_NO
      T_PUSH : Bool := false;   // Habilitar conmutación de transición en modo semiautomático
   END_VAR
   VAR_OUTPUT
      InicioEmergencia : Bool;
      InitGrafcets : Bool;
      ResetGrafcets : Bool;
      S_NO : Int := 0;   // Número de etapa
      S_MORE : Bool := false;   // Existen más etapas que pueden mostrarse en S_NO.
      S_ACTIVE : Bool := false;   // El incremento presente en el parámetro S_NO está activo
      ERR_FLT : Bool := false;   // Error de grupo interlock o supervisión
      AUTO_ON : Bool := false;   // Modo automático activado
      TAP_ON : Bool := false;   // Modo semiautomático/etapa con transición activada
      TOP_ON : Bool := false;   // Modo semiautomático/Ignorar transición activado
      MAN_ON : Bool := false;   // Modo manual activado
   END_VAR
   VAR
      HMI_INFO : Array[0..10] of UInt;
      IF_PAR : G7_IfParPlus_V4;
      RT_DATA : G7_RTDataPlus_V4;   // Área de datos interna
      Trans1 : G7_TransitionPlus_V4;   // Estructura de la transición
      Trans2 : G7_TransitionPlus_V4;   // Estructura de la transición
      Trans3 : G7_TransitionPlus_V4;   // Estructura de la transición
      Trans4 : G7_TransitionPlus_V4;   // Estructura de la transición
      Trans5 : G7_TransitionPlus_V4;   // Estructura de la transición
      X800 : G7_StepPlus_V4;   // Estructura de la etapa
      "801" : G7_StepPlus_V4;   // Estructura de la etapa
      "802" : G7_StepPlus_V4;   // Estructura de la etapa
      "803" : G7_StepPlus_V4;   // Estructura de la etapa
      X805 : G7_StepPlus_V4;   // Estructura de la etapa
      "804" : G7_StepPlus_V4;   // Estructura de la etapa
      SINI : Array[0..3] of USInt;
      LSTT : Array[0..4] of USInt;
      ATAJ : Array[0..4] of USInt;
      ATAB : Array[0..4] of USInt;
      PSTT : Array[0..4] of USInt;
      NSTT : Array[0..4] of USInt;
      ASSJ : Array[0..5] of USInt;
      ASSB : Array[0..5] of USInt;
      PTTS : Array[0..5] of USInt;
      NTTS : Array[0..5] of USInt;
      SW_SQTS : Array[0..5] of USInt;
      SWITCH : Array[0..1] of USInt;
      TVX : Array[0..3] of USInt;
      TTX : Array[0..3] of USInt;
      TSX : Array[0..3] of USInt;
      S00X : Array[0..3] of USInt;
      SOFFX : Array[0..3] of USInt;
      SONX : Array[0..3] of USInt;
      SAX : Array[0..3] of USInt;
      SERRX : Array[0..6] of USInt;
      SMX : Array[0..6] of USInt;
      S0X : Array[0..6] of USInt;
      S1X : Array[0..6] of USInt;
      IL_ALARM_INST : Diag_Alarm;
      SUP_ALARM_INST : Diag_Alarm;
      STEP_TIME_ALARM_INST : Diag_Alarm;
      IEC_TIMER_INST : IEC_TIMER;
      TRANSACTION_FLAG : Bool := false;
   END_VAR
   // SINI[0] := 2;
   // SINI[2] := 255;
   // SINI[3] := 255;
   // LSTT[0] := 255;
   // LSTT[1] := 255;
   // LSTT[2] := 255;
   // LSTT[3] := 255;
   // ATAJ[1] := 1;
   // ATAJ[2] := 2;
   // ATAJ[3] := 3;
   // ATAJ[4] := 4;
   // ATAB[1] := 1;
   // ATAB[2] := 2;
   // ATAB[3] := 3;
   // ATAB[4] := 4;
   // PSTT[1] := 1;
   // PSTT[2] := 2;
   // PSTT[3] := 3;
   // PSTT[4] := 4;
   // NSTT[0] := 1;
   // NSTT[1] := 2;
   // NSTT[2] := 4;
   // NSTT[3] := 5;
   // ASSJ[1] := 1;
   // ASSJ[2] := 5;
   // ASSJ[3] := 3;
   // ASSJ[4] := 4;
   // ASSJ[5] := 2;
   // ASSB[1] := 3;
   // ASSB[2] := 2;
   // ASSB[3] := 1;
   // ASSB[4] := 4;
   // ASSB[5] := 5;
   // PTTS[0] := 255;
   // PTTS[2] := 1;
   // PTTS[4] := 2;
   // PTTS[5] := 3;
   // NTTS[1] := 1;
   // NTTS[2] := 2;
   // NTTS[3] := 3;
   // NTTS[4] := 4;
   // NTTS[5] := 2;
   // SW_SQTS[1] := 1;
   // SW_SQTS[2] := 1;
   // SW_SQTS[3] := 2;
   // SW_SQTS[4] := 3;
   // SW_SQTS[5] := 2;
   // SWITCH[0] := 64;
   // SWITCH[1] := 2;
   // TVX[0] := 16#1;
   // TTX[0] := 16#1;
   // TSX[0] := 16#1;
   // S00X[0] := 16#1;
   // SOFFX[0] := 16#1;
   // SONX[0] := 16#1;
   // SAX[0] := 16#1;
   // SERRX[0] := 16#1;
   // SMX[0] := 16#1;
   // S0X[0] := 16#1;
   // S1X[0] := 16#1;
BEGIN
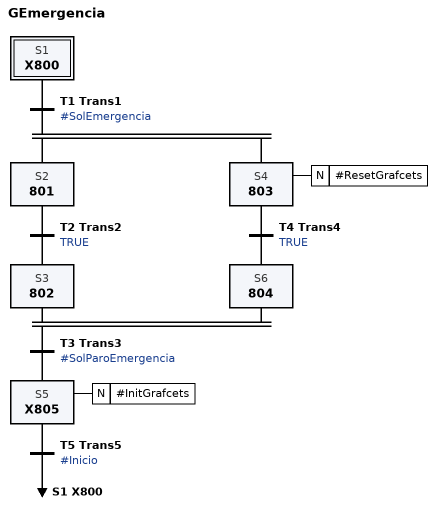
   // sequencer 1
   INITIAL_STEP X800:   // S1, max time T#10S, warning time T#7S
   END_STEP
   TRANSITION Trans1 FROM X800 TO ("801", "803")   // T1
      := #SolEmergencia;
   END_TRANSITION
   STEP "801":   // S2, max time T#10S, warning time T#7S
   END_STEP
   TRANSITION Trans2 FROM "801" TO "802"   // T2
      := TRUE;
   END_TRANSITION
   STEP "802":   // S3, max time T#10S, warning time T#7S
   END_STEP
   STEP "803":   // S4, max time T#10S, warning time T#7S
              N    #ResetGrafcets
   END_STEP
   TRANSITION Trans4 FROM "803" TO "804"   // T4
      := TRUE;
   END_TRANSITION
   STEP X805:   // S5, max time T#10S, warning time T#7S
              N    #InitGrafcets
   END_STEP
   TRANSITION Trans5 FROM X805 TO X800   // T5, jump
      := #Inicio;
   END_TRANSITION
   STEP "804":   // S6, max time T#10S, warning time T#7S
   END_STEP
   TRANSITION Trans3 FROM ("802", "804") TO X805   // T3
      := #SolParoEmergencia;
   END_TRANSITION
END_FUNCTION_BLOCK

ORGANIZATION_BLOCK "Main"   // OB1, LAD, ProgramCycle
TITLE = "Main Program Sweep (Cycle)"
{ S7_Optimized_Access := 'TRUE' }
VERSION : 0.1
   VAR_INPUT
      Initial_Call : Bool;   // Initial call of this OB
      Remanence : Bool;   // =True, if remanent data are available
   END_VAR
   VAR_TEMP
      Indice : Int;
   END_VAR
   VAR_TEMP   // added for the SCL form of the ladder/FBD networks
      _w1 : Bool;
      _w2 : Bool;
   END_VAR
BEGIN

REGION Network 1: Instancias FBs
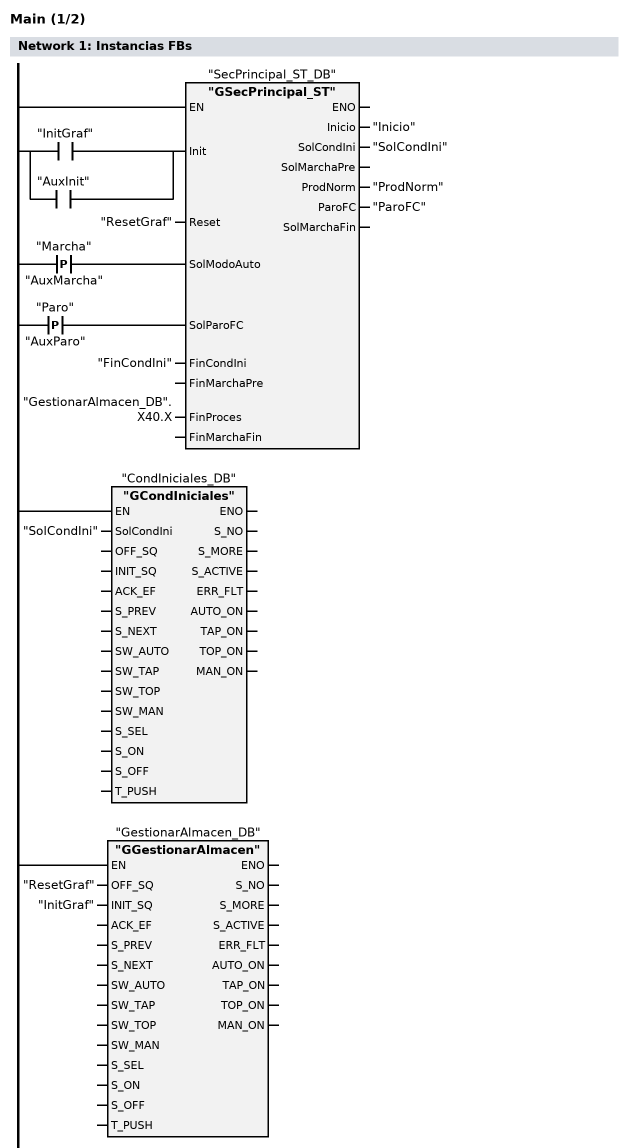
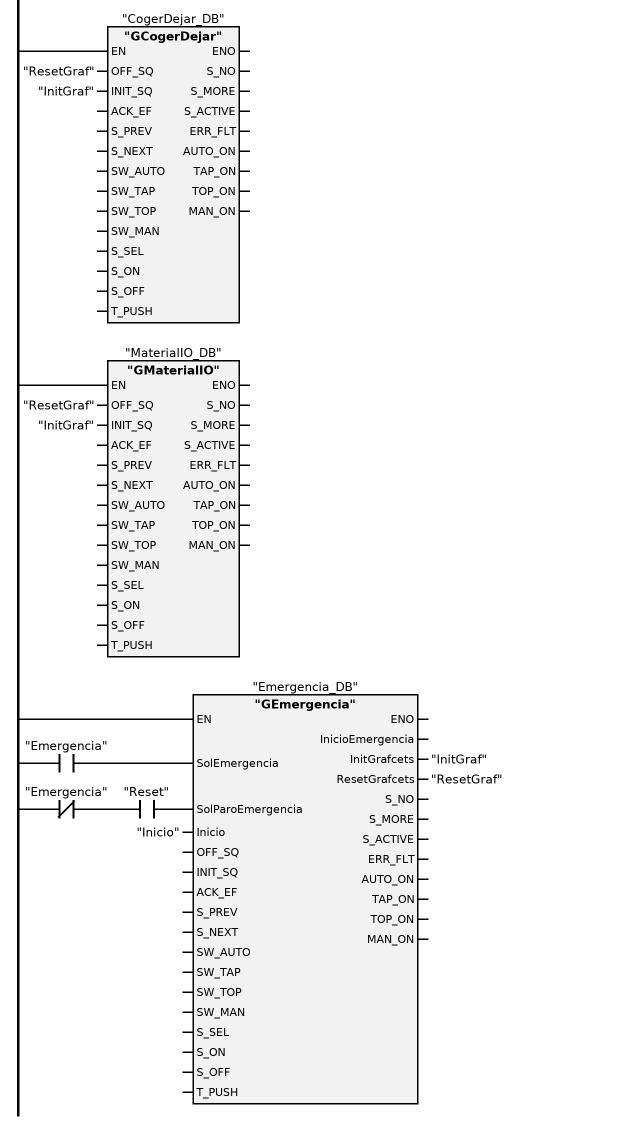
   RUNG wire#powerrail
      "SecPrincipal_ST_DB"(Init := wire#w1, SolModoAuto := wire#w2, SolParoFC := wire#w3, Reset := "ResetGraf", FinCondIni := "FinCondIni", FinMarchaPre :=, FinProces := "GestionarAlmacen_DB".X40.X, FinMarchaFin :=, Inicio => "Inicio", SolCondIni => "SolCondIni", SolMarchaPre =>, ProdNorm => "ProdNorm", ParoFC => "ParoFC", SolMarchaFin =>)
   END_RUNG
   RUNG wire#powerrail
      Contact( "InitGraf" )
   END_RUNG wire#w1
   RUNG wire#powerrail
      Contact( "AuxInit" )
   END_RUNG wire#w1
   RUNG wire#powerrail
      P_Contact(operand := "Marcha", bit := "AuxMarcha")
   END_RUNG wire#w2
   RUNG wire#powerrail
      P_Contact(operand := "Paro", bit := "AuxParo")
   END_RUNG wire#w3
   RUNG wire#powerrail
      "CondIniciales_DB"(SolCondIni := "SolCondIni", OFF_SQ :=, INIT_SQ :=, ACK_EF :=, S_PREV :=, S_NEXT :=, SW_AUTO :=, SW_TAP :=, SW_TOP :=, SW_MAN :=, S_SEL :=, S_ON :=, S_OFF :=, T_PUSH :=, S_NO =>, S_MORE =>, S_ACTIVE =>, ERR_FLT =>, AUTO_ON =>, TAP_ON =>, TOP_ON =>, MAN_ON =>)
   END_RUNG
   RUNG wire#powerrail
      "GestionarAlmacen_DB"(OFF_SQ := "ResetGraf", INIT_SQ := "InitGraf", ACK_EF :=, S_PREV :=, S_NEXT :=, SW_AUTO :=, SW_TAP :=, SW_TOP :=, SW_MAN :=, S_SEL :=, S_ON :=, S_OFF :=, T_PUSH :=, S_NO =>, S_MORE =>, S_ACTIVE =>, ERR_FLT =>, AUTO_ON =>, TAP_ON =>, TOP_ON =>, MAN_ON =>)
   END_RUNG
   RUNG wire#powerrail
      "CogerDejar_DB"(OFF_SQ := "ResetGraf", INIT_SQ := "InitGraf", ACK_EF :=, S_PREV :=, S_NEXT :=, SW_AUTO :=, SW_TAP :=, SW_TOP :=, SW_MAN :=, S_SEL :=, S_ON :=, S_OFF :=, T_PUSH :=, S_NO =>, S_MORE =>, S_ACTIVE =>, ERR_FLT =>, AUTO_ON =>, TAP_ON =>, TOP_ON =>, MAN_ON =>)
   END_RUNG
   RUNG wire#powerrail
      "MaterialIO_DB"(OFF_SQ := "ResetGraf", INIT_SQ := "InitGraf", ACK_EF :=, S_PREV :=, S_NEXT :=, SW_AUTO :=, SW_TAP :=, SW_TOP :=, SW_MAN :=, S_SEL :=, S_ON :=, S_OFF :=, T_PUSH :=, S_NO =>, S_MORE =>, S_ACTIVE =>, ERR_FLT =>, AUTO_ON =>, TAP_ON =>, TOP_ON =>, MAN_ON =>)
   END_RUNG
   RUNG wire#powerrail
      "Emergencia_DB"(SolEmergencia := wire#w4, SolParoEmergencia := wire#w5, Inicio := "Inicio", OFF_SQ :=, INIT_SQ :=, ACK_EF :=, S_PREV :=, S_NEXT :=, SW_AUTO :=, SW_TAP :=, SW_TOP :=, SW_MAN :=, S_SEL :=, S_ON :=, S_OFF :=, T_PUSH :=, InicioEmergencia =>, InitGrafcets => "InitGraf", ResetGrafcets => "ResetGraf", S_NO =>, S_MORE =>, S_ACTIVE =>, ERR_FLT =>, AUTO_ON =>, TAP_ON =>, TOP_ON =>, MAN_ON =>)
   END_RUNG
   RUNG wire#powerrail
      Contact( "Emergencia" )
   END_RUNG wire#w4
   RUNG wire#powerrail
      I_Contact( "Emergencia" )
      Contact( "Reset" )
   END_RUNG wire#w5
   // the same network as SCL:
   #_w1 := "Marcha" AND NOT "AuxMarcha";   // rising edge of "Marcha"
   "AuxMarcha" := "Marcha";
   #_w2 := "Paro" AND NOT "AuxParo";   // rising edge of "Paro"
   "AuxParo" := "Paro";
   "SecPrincipal_ST_DB"(Init := "InitGraf" OR "AuxInit",   // "GSecPrincipal_ST"
                        Reset := "ResetGraf",
                        SolModoAuto := #_w1,
                        SolParoFC := #_w2,
                        FinCondIni := "FinCondIni",
                        FinProces := "GestionarAlmacen_DB".X40.X,
                        Inicio => "Inicio",
                        SolCondIni => "SolCondIni",
                        ProdNorm => "ProdNorm",
                        ParoFC => "ParoFC");
   "CondIniciales_DB"(SolCondIni := "SolCondIni");   // "GCondIniciales"
   "GestionarAlmacen_DB"(OFF_SQ := "ResetGraf", INIT_SQ := "InitGraf");   // "GGestionarAlmacen"
   "CogerDejar_DB"(OFF_SQ := "ResetGraf", INIT_SQ := "InitGraf");   // "GCogerDejar"
   "MaterialIO_DB"(OFF_SQ := "ResetGraf", INIT_SQ := "InitGraf");   // "GMaterialIO"
   "Emergencia_DB"(SolEmergencia := "Emergencia",   // "GEmergencia"
                   SolParoEmergencia := NOT "Emergencia" AND "Reset",
                   Inicio := "Inicio",
                   InitGrafcets => "InitGraf",
                   ResetGrafcets => "ResetGraf");
END_REGION

REGION Network 2: Indicar el destino del elevador
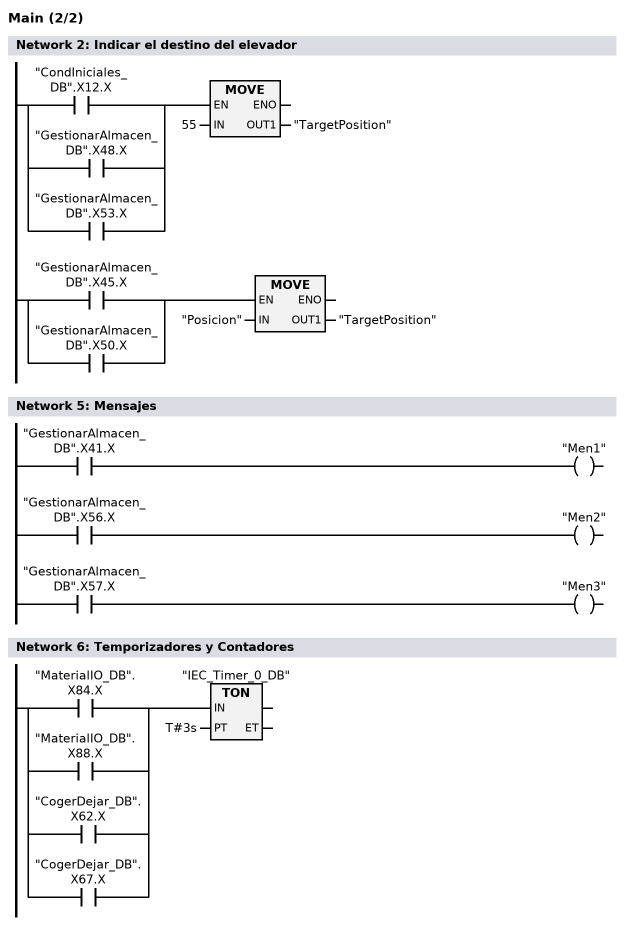
   RUNG wire#powerrail
      Contact( "CondIniciales_DB".X12.X )
      wire#w1
      Move(in := 55, out1 => "TargetPosition")
   END_RUNG
   RUNG wire#powerrail
      Contact( "GestionarAlmacen_DB".X48.X )
   END_RUNG wire#w1
   RUNG wire#powerrail
      Contact( "GestionarAlmacen_DB".X53.X )
   END_RUNG wire#w1
   RUNG wire#powerrail
      Contact( "GestionarAlmacen_DB".X45.X )
      wire#w2
      Move(in := "Posicion", out1 => "TargetPosition")
   END_RUNG
   RUNG wire#powerrail
      Contact( "GestionarAlmacen_DB".X50.X )
   END_RUNG wire#w2
   // the same network as SCL:
   IF "CondIniciales_DB".X12.X OR "GestionarAlmacen_DB".X48.X OR "GestionarAlmacen_DB".X53.X THEN
       "TargetPosition" := 55;
   END_IF;
   IF "GestionarAlmacen_DB".X45.X OR "GestionarAlmacen_DB".X50.X THEN "TargetPosition" := "Posicion"; END_IF;
END_REGION

REGION Network 3 (SCL): Inicializar todos los elementos del array AlmacenOcupación a cero (almacén libre)
   IF "InicializarAlmacenOcupacion" THEN
       FOR #Indice := 1 TO 54 DO
           "Sensores".AlmacenOcupacion[#Indice] := 0;
       END_FOR;
       #Indice := 1;
   END_IF;
END_REGION

REGION Network 4 (STL)
         A     "InicializarAlmacenOcupacion";
         JCN   EXIT;

         OPN   "Sensores";
         LAR1  P#0.0;

         L     54;
   FOR:  T     #Indice;

         CLR;
         =     DBX[AR1,P#0.0];

         +AR1  P#0.1;

         L     #Indice;
         LOOP  FOR;

   EXIT: NOP   0;
END_REGION

REGION Network 5: Mensajes
   RUNG wire#powerrail
      Contact( "GestionarAlmacen_DB".X41.X )
      Coil( "Men1" )
   END_RUNG
   RUNG wire#powerrail
      Contact( "GestionarAlmacen_DB".X56.X )
      Coil( "Men2" )
   END_RUNG
   RUNG wire#powerrail
      Contact( "GestionarAlmacen_DB".X57.X )
      Coil( "Men3" )
   END_RUNG
   // the same network as SCL:
   "Men1" := "GestionarAlmacen_DB".X41.X;
   "Men2" := "GestionarAlmacen_DB".X56.X;
   "Men3" := "GestionarAlmacen_DB".X57.X;
END_REGION

REGION Network 6: Temporizadores y Contadores
   "IEC_Timer_0_DB".TON(IN := "MaterialIO_DB".X84.X OR "MaterialIO_DB".X88.X OR "CogerDejar_DB".X62.X OR "CogerDejar_DB".X67.X,
                        PT := T#3s);
END_REGION
END_ORGANIZATION_BLOCK

(* ===== HMI "HMI_RT_1" =====
system functions are stored by id; their names below are inferred from use
connection "HMI_Conexión_1": ETHERNET, SMART_S7_1500_OMS

HMI tags "Tabla de variables estándar"
   "Número_imagen_variable" : UInt, internal

HMI tags "Tabla de variables estándar_1"
   "Marcha" : Bool = PLC Marcha AT %M5.0, 1 s
   "Paro" : Bool = PLC Paro AT %M5.1, 1 s
   "Posicion" : Int = PLC Posicion AT %MW8, 1 s
   "Reset" : Bool = PLC Reset AT %M5.2, 1 s
   "DejarCoger" : Bool = PLC DejarCoger AT %M0.5, 1 s
   "Sensores_AlmacenOcupacion19" : Bool = PLC Sensores.AlmacenOcupacion[19] AT %DB1.DBX2.2, 1 s
   "Sensores_AlmacenOcupacion1" : Bool = PLC Sensores.AlmacenOcupacion[1] AT %DB1.DBX0.0, 1 s
   "Sensores_AlmacenOcupacion10" : Bool = PLC Sensores.AlmacenOcupacion[10] AT %DB1.DBX1.1, 1 s
   "Sensores_AlmacenOcupacion2" : Bool = PLC Sensores.AlmacenOcupacion[2] AT %DB1.DBX0.1, 1 s
   "Sensores_AlmacenOcupacion3" : Bool = PLC Sensores.AlmacenOcupacion[3] AT %DB1.DBX0.2, 1 s
   "Sensores_AlmacenOcupacion4" : Bool = PLC Sensores.AlmacenOcupacion[4] AT %DB1.DBX0.3, 1 s
   "Sensores_AlmacenOcupacion11" : Bool = PLC Sensores.AlmacenOcupacion[11] AT %DB1.DBX1.2, 1 s
   "Sensores_AlmacenOcupacion12" : Bool = PLC Sensores.AlmacenOcupacion[12] AT %DB1.DBX1.3, 1 s
   "Sensores_AlmacenOcupacion13" : Bool = PLC Sensores.AlmacenOcupacion[13] AT %DB1.DBX1.4, 1 s
   "Sensores_AlmacenOcupacion14" : Bool = PLC Sensores.AlmacenOcupacion[14] AT %DB1.DBX1.5, 1 s
   "Sensores_AlmacenOcupacion20" : Bool = PLC Sensores.AlmacenOcupacion[20] AT %DB1.DBX2.3, 1 s
   "Sensores_AlmacenOcupacion21" : Bool = PLC Sensores.AlmacenOcupacion[21] AT %DB1.DBX2.4, 1 s
   "Sensores_AlmacenOcupacion22" : Bool = PLC Sensores.AlmacenOcupacion[22] AT %DB1.DBX2.5, 1 s
   "Sensores_AlmacenOcupacion32" : Bool = PLC Sensores.AlmacenOcupacion[32] AT %DB1.DBX3.7, 1 s
   "Inicio" : Bool = PLC Inicio AT %M0.0, 1 s
   "SolCondIni" : Bool = PLC SolCondIni AT %M0.1, 1 s
   "ProdNorm" : Bool = PLC ProdNorm AT %M0.3, 1 s
   "ParoFC" : Bool = PLC ParoFC AT %M0.4, 1 s
   "Emergencia" : Bool = PLC Emergencia AT %M10.3, 1 s
   "AuxInit" : Bool = PLC AuxInit AT %M2.0, 1 s
   "Sensores_AlmacenOcupacion5" : Bool = PLC Sensores.AlmacenOcupacion[5] AT %DB1.DBX0.4, 1 s
   "Sensores_AlmacenOcupacion31" : Bool = PLC Sensores.AlmacenOcupacion[31] AT %DB1.DBX3.6, 1 s
   "Sensores_AlmacenOcupacion30" : Bool = PLC Sensores.AlmacenOcupacion[30] AT %DB1.DBX3.5, 1 s
   "Sensores_AlmacenOcupacion29" : Bool = PLC Sensores.AlmacenOcupacion[29] AT %DB1.DBX3.4, 1 s
   "Sensores_AlmacenOcupacion28" : Bool = PLC Sensores.AlmacenOcupacion[28] AT %DB1.DBX3.3, 1 s
   "Sensores_AlmacenOcupacion23" : Bool = PLC Sensores.AlmacenOcupacion[23] AT %DB1.DBX2.6, 1 s
   "AuxInit(1)" : Bool = PLC AuxInit AT %M2.0, 1 s
   "AuxInit(2)" : Bool = PLC AuxInit AT %M2.0, 1 s

text list "Nombre_imagen_lista_texto": 1 'Imagen raíz'

Template "Plantilla_1" 480x272
   Button "Salir" at 388,227 size 63x44; TextOff 'Salir'; PictureOff "ExitRuntime_KTP400_Basic_PN_TR"; PictureOn "ExitRuntime_KTP400_Basic_PN_TR"
      on Release: StopRuntime(0)
   Button "Template_Button" at 268,227 size 63x44; TextOff 'Text'
   Button "Avisos" at 148,227 size 63x44; TextOff 'Avisos'; PictureOff "AlarmDisplay_KTP400_Basic_PN_TR"; PictureOn "AlarmDisplay_KTP400_Basic_PN_TR"
      on Release: function_ef3f5d25("Ventana de avisos_no_acusado", -1)
   Button "Imagen inicial" at 28,227 size 63x44; TextOff 'Imagen inicial'; PictureOff "NavigateHome_KTP400_Basic_PN_TR"; PictureOn "NavigateHome_KTP400_Basic_PN_TR"
      on Release: ActivateScreen("Imagen raíz", 0)
   SymbolicIOField "Imagen_campo_ES_simbólico" at 82,8 size 311x29; TextOff '0'; TextOn '1'; TextList "Nombre_imagen_lista_texto"
      ProcessValue <- "Número_imagen_variable"
      on Change: ActivateScreenByNumber("Número_imagen_variable", 0)
   DateTimeField "HmiScreenItemData" at 395,22 size 85x22
   DateTimeField "HmiScreenItemData_1" at 395,0 size 85x22
   GraphicView "Logotipo" at 0,0 size 80x45; Picture "Logotipo de HMI_1"

screen "Imagen raíz" 480x272, template "Plantilla_1"
   Rectangle "Rectángulo_1" at 162,52 size 42x36
      Appearance <- "Sensores_AlmacenOcupacion32"
   Rectangle "Rectángulo_3" at 203,52 size 42x36
      Appearance <- "Sensores_AlmacenOcupacion31"
   Rectangle "Rectángulo_2" at 244,52 size 42x36
      Appearance <- "Sensores_AlmacenOcupacion30"
   Rectangle "Rectángulo_4" at 285,52 size 42x36
      Appearance <- "Sensores_AlmacenOcupacion29"
   Rectangle "Rectángulo_5" at 326,52 size 42x36
      Appearance <- "Sensores_AlmacenOcupacion28"
   Rectangle "Rectángulo_6" at 162,88 size 42x36
      Appearance <- "Sensores_AlmacenOcupacion23"
   Rectangle "Rectángulo_7" at 203,88 size 42x36
      Appearance <- "Sensores_AlmacenOcupacion22"
   Rectangle "Rectángulo_8" at 244,88 size 42x36
      Appearance <- "Sensores_AlmacenOcupacion21"
   Rectangle "Rectángulo_9" at 285,88 size 42x36
      Appearance <- "Sensores_AlmacenOcupacion20"
   Rectangle "Rectángulo_10" at 326,88 size 42x36
      Appearance <- "Sensores_AlmacenOcupacion19"
   Rectangle "Rectángulo_11" at 162,124 size 42x36
      Appearance <- "Sensores_AlmacenOcupacion14"
   Rectangle "Rectángulo_12" at 203,124 size 42x36
      Appearance <- "Sensores_AlmacenOcupacion13"
   Rectangle "Rectángulo_13" at 244,124 size 42x36
      Appearance <- "Sensores_AlmacenOcupacion12"
   Rectangle "Rectángulo_14" at 285,124 size 42x36
      Appearance <- "Sensores_AlmacenOcupacion11"
   Rectangle "Rectángulo_15" at 326,124 size 42x36
      Appearance <- "Sensores_AlmacenOcupacion10"
   Rectangle "Rectángulo_16" at 162,160 size 42x36
      Appearance <- "Sensores_AlmacenOcupacion5"
   Rectangle "Rectángulo_17" at 203,160 size 42x36
      Appearance <- "Sensores_AlmacenOcupacion4"
   Rectangle "Rectángulo_18" at 244,160 size 42x36
      Appearance <- "Sensores_AlmacenOcupacion3"
   Rectangle "Rectángulo_19" at 285,160 size 42x36
      Appearance <- "Sensores_AlmacenOcupacion2"
   Rectangle "Rectángulo_20" at 326,160 size 42x36
      Appearance <- "Sensores_AlmacenOcupacion1"
   Button "Botón_6" at 174,153 size 18x12; TextOff '14'
   Button "Botón_7" at 214,153 size 18x12; TextOff '13'
   Button "Botón_8" at 254,153 size 18x12; TextOff '12'
   Button "Botón_9" at 294,153 size 18x12; TextOff '11'
   Button "Botón_10" at 335,153 size 18x12; TextOff '10'
   Button "Botón_11" at 174,117 size 18x12; TextOff '23'
   Button "Botón_12" at 214,117 size 18x12; TextOff '22'
   Button "Botón_13" at 255,117 size 18x12; TextOff '21'
   Button "Botón_14" at 295,117 size 18x12; TextOff '20'
   Button "Botón_15" at 336,117 size 18x12; TextOff '19'
   Button "Botón_16" at 174,82 size 18x12; TextOff '32'
   Button "Botón_17" at 214,82 size 18x12; TextOff '31'
   Button "Botón_18" at 255,82 size 18x12; TextOff '30'
   Button "Botón_19" at 295,82 size 18x12; TextOff '29'
   Button "Botón_20" at 336,82 size 18x12; TextOff '28'
   Button "Botón_1" at 174,189 size 18x12; TextOff '05'
   Button "Botón_2" at 214,189 size 18x12; TextOff '04'
   Button "Botón_3" at 255,189 size 18x12; TextOff '03'
   Button "Botón_4" at 295,189 size 18x12; TextOff '02'
   Button "Botón_5" at 336,189 size 18x12; TextOff '01'
   TextField "HmiScreenItemData_7" at 209,0 size 80x22; Text 'Posición'
   IOField "Campo ES_2" at 232,21 size 30x24; FormatPattern 99
      ProcessValue <- "Posicion"
   Button "Botón_21" at 12,12 size 66x30; TextOff 'Marcha'
      on Release: ResetBit("Marcha")
      on Press: SetBit("Marcha")
      Appearance <- "Marcha"
   Button "Botón_22" at 12,48 size 66x30; TextOff 'Paro'
      on Release: ResetBit("Paro")
      on Press: SetBit("Paro")
      Appearance <- "Paro"
   Button "Botón_23" at 12,85 size 66x30; TextOff 'Reset'
      on Release: ResetBit("Reset")
      on Press: SetBit("Reset")
      Appearance <- "Reset"
   Switch "Interruptor_1" at 282,24 size 84x18; TextOn 'Dejar'; CaptionText 'Switch'; TextOff 'Coger'
      ProcessValue <- "DejarCoger"
   Button "Botón_24" at 12,186 size 90x30; TextOff 'Emergencia'
      on Release: ResetBit("Emergencia")
      on Press: SetBit("Emergencia")
      Appearance <- "Emergencia"
   Circle "Círculo_1" at 391,12 size 12x12
      Appearance <- "Inicio"
   TextField "Campo de texto_1" at 404,10 size 32x15; Text 'Inicio'
   Circle "Círculo_2" at 391,26 size 12x12
      Appearance <- "SolCondIni"
   TextField "Campo de texto_2" at 404,24 size 74x15; Text 'Cond Iniciales'
   Circle "Círculo_3" at 391,41 size 12x12
      Appearance <- "ProdNorm"
   Circle "Círculo_4" at 391,56 size 12x12
      Appearance <- "ParoFC"
   TextField "Campo de texto_3" at 404,39 size 70x15; Text 'Prod. Normal'
   TextField "Campo de texto_4" at 404,54 size 44x15; Text 'Paro FC'
   Button "Botón_25" at 408,78 size 60x24; TextOff 'AuxInit'
      on Release: ResetBit("AuxInit")
      on Press: SetBit("AuxInit")
      Appearance <- "AuxInit"
*)